// TwinCAT 3 PLC project TwinCAT_3_Program
// ProgramVersion: 3.1.4024.0
// libraries:
//   CmpBitmapPool, * (System)
//   Recipe Management, * (System)
//   Tc2_ControllerToolbox, * (Beckhoff Automation GmbH)
//   Tc2_Drive, * (Beckhoff Automation GmbH)
//   Tc2_EtherCAT, * (Beckhoff Automation GmbH)
//   Tc2_IoFunctions, * (Beckhoff Automation GmbH)
//   Tc2_Math, * (Beckhoff Automation GmbH)
//   Tc2_MC2, * (Beckhoff Automation GmbH)
//   Tc2_MC2_Drive, * (Beckhoff Automation GmbH)
//   Tc2_ModbusRTU, * (Beckhoff Automation GmbH)
//   Tc2_ModbusSrv, * (Beckhoff Automation GmbH)
//   Tc2_SerialCom, * (Beckhoff Automation GmbH)
//   Tc2_Standard, * (Beckhoff Automation GmbH)
//   Tc2_SUPS, * (Beckhoff Automation GmbH)
//   Tc2_System, * (Beckhoff Automation GmbH)
//   Tc2_Utilities, * (Beckhoff Automation GmbH)
//   Tc2_XmlDataSrv, * (Beckhoff Automation GmbH)
//   Tc3_Module, * (Beckhoff Automation GmbH)
//   VisuDialogs, * (System)
//   VisuSymbols,3.5.10.0,System
// project tree:
//   DUTs/DS TBD/ DSA1_ArmHorzPosInput.TcDUT, DSA1_ArmHorzPosOutput.TcDUT, DSA1_ArmPnpSequenceCall.TcDUT, DSA1_fbPnpSequenceMemoryCall.TcDUT, DSA1_fbPnpSequenceMemoryStore.TcDUT, DSA1_PnpSequenceMemory.TcDUT, DSA1_UpDownMovement.TcDUT, DSA21_UpDownPatternCall.TcDUT, DSA21_UpDownPatternMemory.TcDUT, DSA21_UpDownPatternStore.TcDUT, DSA31_ArmSpeedProfileCall.TcDUT, DSA31_ArmSpeedProfileMemory.TcDUT, DSA31_ArmSpeedProfileStore.TcDUT, DSA32_StationZoneHeight.TcDUT, DSA32_StationZoneHeightIntNotInUsed.TcDUT, DSA32_StationZonePosOut.TcDUT, DSChemicalWithoutDosingPump.TcDUT, DSGnr_CalledArmPnpParameter.TcDUT, DSPnpAgitationParameter.TcDUT, DSV2_A1_ArmHorzPosInput.TcDUT, DSV2_A1_ArmHorzPosOutput.TcDUT, DSV2_A1_ArmPnpSequenceCall.TcDUT, DSV2_A1_fbPnpSequenceMemoryCall.TcDUT, DSV2_A1_fbPnpSequenceMemoryStore.TcDUT, DSV2_A1_PnpSequenceMemory.TcDUT, DSV2_ApolloRemoteHoistInput.TcDUT, DSV2_ApolloRemoteHoistOutput.TcDUT, DSV2_ArmPosition.TcDUT, DSV2_BasketInfo.TcDUT, DSV2_ClangsonicGenerator.TcDUT, DSV2_fbGnrProductRecipeMemoryOut.TcDUT, DSV2_fbStationSequenceRecipeCall.TcDUT, DSV2_fbStationSequenceRecipeStore.TcDUT, DSV2_Gnr_CalledArmPnpParameter.TcDUT, DSV2_MinMaxEffTime.TcDUT, DSV2_ModbusControl.TcDUT, DSV2_SSERSourceMinMaxTime.TcDUT, DSV2_StationSequenceRecipeMemory.TcDUT, DSV2_StnMinMaxEffTIme.TcDUT, DSV2_TimeTrackerInput.TcDUT, DSV3_BarcodeRegistration.TcDUT, DSV3_JRS_Alarm.TcDUT, DSV3_JRS_HMI.TcDUT, DSV3_JRS_Input.TcDUT, DSV3_JRS_Output.TcDUT, DSV3_StnInterlock.TcDUT, DSV3_TempCtrlParameter.TcDUT, DSV3_TempCtrlRecipe.TcDUT, DSV3_XML_Recipe.TcDUT, DS_ArmPnPInOut.TcDUT, DS_BasketInfo.TcDUT, DS_BrensonEnclosure.TcDUT, DS_BrensonGenerator.TcDUT, DS_BrensonMulFreqSwitching.TcDUT, DS_ClangsonicGenerator.TcDUT, DS_fbGnrProductRecipeMemoryOut.TcDUT, DS_fbStationSequenceRecipeCall.TcDUT, DS_fbStationSequenceRecipeStore.TcDUT, DS_fbStationSubRecipeCall.TcDUT, DS_fbStationSubRecipeStore.TcDUT, DS_fbStnSeqProcessCtrl.TcDUT, DS_HMIStationDisplayInfo.TcDUT, DS_HomingSetting.TcDUT, DS_Inverter.TcDUT, DS_ProminentDosingHMI.TcDUT, DS_SA_Movement.TcDUT, DS_Servo.TcDUT, DS_StationSequenceRecipeMemory.TcDUT, DS_StnSeqProInput.TcDUT, DS_StnSeqProOutput.TcDUT, DS_SubRecipeMemory.TcDUT, DS_TimeTrackerInput.TcDUT, DS_WeberEnclosure.TcDUT, DS_WeberGenerator.TcDUT, DS_WeberMulFreqSwitching.TcDUT, DS_XMLRW.TcDUT, DS_XML_InputOutput.TcDUT, En_LogFileType.TcDUT, En_TimeInterval.TcDUT
//   DUTs/DS Twincat 3/Barcode/ DS_SerialCommunication.TcDUT
//   DUTs/DS Twincat 3/CSV/ DS_CsvErrorLog.TcDUT, DS_CsvLog.TcDUT, DS_CsvReport.TcDUT, E_CsvActionType.TcDUT
//   DUTs/DS Twincat 3/ DS_HMI_MappingVariable.TcDUT, DS_LocalSystemTime.TcDUT, DS_XML_Persistent_Analog.TcDUT, DS_XML_Persistent_Arm.TcDUT, DS_XML_Persistent_Barcode.TcDUT, DS_XML_Persistent_Deactivate.TcDUT, DS_XML_Persistent_Digital.TcDUT, DS_XML_Persistent_Memory.TcDUT, DS_XML_Persistent_Process.TcDUT, DS_XML_Persistent_SevenDay.TcDUT, DS_XML_Persistent_TimeOptimize.TcDUT, E_HmiLanguage.TcDUT, ST_DataLog.TcDUT
//   DUTs/DS Twincat 3/Enum/ Digital_Input.TcDUT, Digital_Output.TcDUT, Enum_Alarm_Others.TcDUT
//   DUTs/DS Twincat 3/Event/ DS_ActiveEventDisplay.TcDUT, DS_Event.TcDUT, DS_EventControl.TcDUT, DS_EventDescriptionCausedRemedy.TcDUT, DS_EventHistory.TcDUT, DS_EventHistoryLogToFile.TcDUT, DS_HistoryEventDisplay.TcDUT, E_EventType.TcDUT
//   DUTs/DS Twincat 3/UserCtrl/ DS_HmiUserReg.TcDUT, DS_HmiUserStatus.TcDUT, DS_VisuElement.TcDUT, eActorType.TcTLEO
//   DUTs/DS Twincat 3/XML/ E_XmlParType.TcDUT, E_XmlRwMode.TcDUT, E_XmlVariableType.TcDUT
//   FBs/B_JKS_CustomFB/fbArmCtrlFolder/ AM_MoveAbsolute.TcPOU, fbArmMoveInterLock.TcPOU, fbArmPnpCtrl.TcPOU, fbAxisPosCtrl.TcPOU, fbGenerateArmPickTransferBit.TcPOU, fbIndMotDecCtrl.TcPOU, fbInverterHorzHome.TcPOU, fbInverterJogCtrl.TcPOU, fbInverterPosCtrl.TcPOU, fbInverterVertHome.TcPOU, fbMotorHomingAxis.TcPOU, fbMultipleArmAgiCtrl.TcPOU, fbServoPosCmp.TcPOU, fbSlowPullAxisCtrl.TcPOU, fb_AxisMovement_Down.TcPOU, fb_AxisMovement_Up.TcPOU, FB_DRIVE_STATUS_ONE_AX.TcPOU
//   FBs/B_JKS_CustomFB/fbBarcodeCtrl/ fbBarcodeScanner.TcPOU, fbBarcodeSorting_10ML5575.TcPOU, fbBarcodeTracer.TcPOU, fbBarcodeTrancerNoCode.TcPOU, fbPreSuffixEliminator.TcPOU
//   FBs/B_JKS_CustomFB/fbConversionCtrl/ AM_InverterConversionHz.TcPOU, fbKeyenceVacSensorTuningkPa.TcPOU, fbRawRatioConversionAllenINV.TcPOU, fbRawRatioConversionReal.TcPOU, fbRawRatioConversionUs.TcPOU, fbRawRatioConversionUsPercent.TcPOU
//   FBs/B_JKS_CustomFB/fbDataLogCtrl/ FB_jx_DataLog.TcPOU, FB_TimeTriggering.TcPOU, FB_WriteLog.TcPOU, F_jx_TS_TO_DATE_STRING.TcPOU, F_jx_TS_TO_DATE_STRING_1.TcPOU, F_jx_TS_TO_TIME_STRING.TcPOU
//   FBs/B_JKS_CustomFB/fbGeneralfbFolder/ fbAssignBadBstCtrl.TcPOU, fbSlidingDoorCtrl.TcPOU, fbToleranceTimeCtrl.TcPOU, UserlevelFB.TcPOU
//   FBs/B_JKS_CustomFB/fbStnDegassingCtrl/ fbStnDegassCtrl.TcPOU
//   FBs/B_JKS_CustomFB/fbUltrasonicCtrl/ BrensonFreqSelector.TcPOU, fbUltrasonicFIFO.TcPOU, fbWeberUS_AI_Conversion.TcPOU, FB_WEBER.TcPOU, WeberFreqSelector.TcPOU
//   FBs/B_JKS_CustomFB/Other/ DoorOpenBasketTransfer.TcPOU, fbConveyorCtrl.TcPOU, fbIndirectAddStringArray.TcPOU, fbKeyConversionBarKpa.TcPOU, fbLdConveyor3Zones.TcPOU, fbLoadingConveyor3Zones.TcPOU, fbMultipleArmBasketMemory.TcPOU, fbPX3524ConversionBarKpa.TcPOU, fbStnRecipeWithSubAndCall.TcPOU, fbUld3ZoneConveyorCtrl.TcPOU, fbUldConveyor3Zones.TcPOU, fb_ArmBasketRotateCtrl.TcPOU, fb_StnCylinderInOutCtrl.TcPOU, HoldingBitSV.TcPOU, ReservoirTankDrain.TcPOU, ReservoirTankDrainNIL.TcPOU, TactTimeFB.TcPOU
//   FBs/B_JKS_NewFB/FBP-AlarmAndEvent/ fbAlarmModule.TcPOU
//   FBs/B_JKS_NewFB/FBP-ArmRelated/ fbA1_ArmHorzPosMemory.TcPOU, fbFBPArmHorzZoneConfirm.TcPOU, fbFBPVertArmPosConfirm.TcPOU, fbGnrProductRecipeMemory.TcPOU
//   FBs/B_JKS_NewFB/FBP-BasketTotalizer/ fbBasketTotalizer.TcPOU, fbStnBasketTotalizer.TcPOU
//   FBs/B_JKS_NewFB/FBP-EncoderIncrementalCtrl/ fbEncoderConversion.TcPOU
//   FBs/B_JKS_NewFB/FBP-HMIAddMapping/ fbHMIAddMappingArrayBool.TcPOU, fbHMIAddMappingArrayInt.TcPOU, fbHMIAddMappingArrayLreal.TcPOU, fbHMIAddMappingArrayReal.TcPOU, fbHMIAddMappingArrayString.TcPOU, fbHMIAddMappingBool.TcPOU, fbHMIAddMappingBoolForManual.TcPOU, fbHMIAddMappingDWordToBoolForManual.TcPOU, fbHMIAddMappingInt.TcPOU, fbHMIAddMappingInt_Word.TcPOU, fbHMIAddMappingLreal.TcPOU, fbHMIAddMappingReal.TcPOU, fbHMIAddMappingReal_Int.TcPOU, fbHMIAddMappingReal_Word.TcPOU, fbHMIAddMappingString.TcPOU
//   FBs/B_JKS_NewFB/FBP-HMI/ fbHMISimulateArmMovement.TcPOU, fbScrMapping.TcPOU
//   FBs/B_JKS_NewFB/FBP-Instrument/ fbBrensonMultiFreqCtrl.TcPOU, fbClangsonicUltrasonic.TcPOU, fbClangsonicUltrasonic_test.TcPOU, fbWeberMultiFreqCtrl.TcPOU
//   FBs/B_JKS_NewFB/FBP-MachineOperationTimeCounter/ fbMachineTimeCounter.TcPOU, fbVacuumPumpTimeCounter.TcPOU
//   FBs/B_JKS_NewFB/FBP-Memory_Sub/ fbA1_PnpSequenceMemory.TcPOU, fbA21_UpDownPattern.TcPOU, fbA31_ArmSpeedProfileMemory.TcPOU, fbA32_MachineZoneHeight.TcPOU, fbA32_StationZoneHeight.TcPOU, fbCallStnSeqSubPro.TcPOU, fbGnrStationMasterController.TcPOU, fbSingleArmBasketMemoryV2.TcPOU, fbStationSequenceRecipe.TcPOU, fbStationSubRecipe.TcPOU, fbStnSeqProcess.TcPOU
//   FBs/B_JKS_NewFB/FBP-ProcessOptimisation/ fbFBPTimeTrackerG2.TcPOU, fbFBPTimeTrackerG3.TcPOU, fbMasterTimeBlockG2.TcPOU, fbRecipeTimeBlockG2.TcPOU, fbTimeBlockSimulatorG2.TcPOU
//   FBs/B_JKS_NewFB/FBP-ProminentDosingPumpCtrl/ fbProminentDosingCtrl.TcPOU
//   FBs/B_JKS_NewFB/FBP-SevenDayAutoOnOff/ fbSevenDaySys.TcPOU
//   FBs/B_JKS_NewFB/FBP-StationRelated/ fbMainStationProcess.TcPOU
//   FBs/B_JKS_NewFB/FBP-TempController/ fbTempControl.TcPOU
//   FBs/B_JKS_NewFB/FBP-TowerLightCtrl/ fbTowerLightCtrl.TcPOU
//   FBs/B_JKS_NewFB_V2/fbArmCtrlFolder/ fbV2_1_ArmPnpCtrl.TcPOU
//   FBs/B_JKS_NewFB_V2/FBP-ArmCtrlFolder/ fbV2_ArmPnpCtrl.TcPOU, fbV2_GenerateArmPickTransferBit.TcPOU
//   FBs/B_JKS_NewFB_V2/FBP-ArmRelated/ fbV2_ArmPosSignalCtrl.TcPOU, fbV2_FBPArmHorzZoneConfirm.TcPOU, fbV2_GnrProductRecipeMemory.TcPOU, NIUfbV2_FBPVertArmPosConfirm.TcPOU
//   FBs/B_JKS_NewFB_V2/FBP-BasketInfoRelated/ fbV2_BasketInfoManager.TcPOU
//   FBs/B_JKS_NewFB_V2/FBP-Function_Sub/ fbAgitationCtrl.TcPOU, fbV2_BasketInfoFinder.TcPOU, fbV2_DSMovementHandler.TcPOU, fbV2_InvAnalogSpdCtrl.TcPOU, fbV2_InvAxisHome.TcPOU, fbV2_InvAxisJog.TcPOU, fbV2_InvPosCtrl.TcPOU
//   FBs/B_JKS_NewFB_V2/FBP-HMI/ fbV2_ScrMapping.TcPOU
//   FBs/B_JKS_NewFB_V2/FBP-Instrument/Dryer/ fbV2_DryerCoolingCtrl.TcPOU (not stored)
//   FBs/B_JKS_NewFB_V2/FBP-LdUldCVRelated/ fbV2_Cv2zonewith2m2sCtrl.TcPOU, fbV2_Cv3zonewith3m3sCtrl.TcPOU, fbV2_Cv4zonewith4m4sCtrl.TcPOU, fbV2_Cv5zonewith5m5sCtrl.TcPOU, fbV2_LdUldCvCtrl.TcPOU
//   FBs/B_JKS_NewFB_V2/FBP-Memory_Sub/ fbV2_A1_PnpSequenceMemory.TcPOU, fbV2_A32_MachineZoneHeight.TcPOU, fbV2_CallStnSeqSubPro.TcPOU, fbV2_GnrStationMasterController.TcPOU, fbV2_SingleArmBasketMemoryV2.TcPOU, fbV2_StationSequenceRecipe.TcPOU, fbV2_StnSeqProcess.TcPOU
//   FBs/B_JKS_NewFB_V2/FBP-MTBSubFB/ fbV2_HMIStnMinMaxEffTimeDisplay.TcPOU, fbV2_MinMaxExtShift.TcPOU, fbV2_SubAnalyzeRTBEffTime.TcPOU, fbV2_SubBusyRTBShifting.TcPOU, fbV2_SubFreeMTBShifting.TcPOU, fbV2_SubMTBFreeSlotGenerator.TcPOU, fbV2_SubMTBRTBCrashCheck.TcPOU, fbV2_SubMTBRunningTime.TcPOU, fbV2_SubRTBBusyLinkMTSUpdate.TcPOU, fbV2_SubRTBEndStepFinder.TcPOU, fbV2_SubRTBGenerateNoCallArmTime.TcPOU, fbV2_SubRTBStnTypeAltIDFinder.TcPOU, fbV2_SubTimeBlockCompare.TcPOU
//   FBs/B_JKS_NewFB_V2/FBP-ProcessOptimisation/ fbV2_FBPTimeTrackerG3.TcPOU, fbV2_MasterTimeBlockG2.TcPOU, fbV2_TimeBlockSimulatorG2.TcPOU
//   FBs/B_JKS_NewFB_V2/FBP-StationRelated/ fbV2_MainStationProcess.TcPOU
//   FBs/B_JKS_NewFB_V2/FBP-TempController/ fbV2_TempControl.TcPOU
//   FBs/B_JKS_NewFB_V3/CSV/ FB3_CsvHandler.TcPOU
//   FBs/B_JKS_NewFB_V3/Event/ FB3_EventModule.TcPOU
//   FBs/B_JKS_NewFB_V3/FBP-Memory_Sub/ fbV3_TemperatureParaRecipe.TcPOU
//   FBs/B_JKS_NewFB_V3/UserCtrl/ FB3_HmiTF1800_UserlevelManagement.TcPOU
//   FBs/B_JKS_NewFB_V3/XML/ FB3_XmlSvrRW_MultipleGVL.TcPOU, FB3_XmlSvrRW_Recipe.TcPOU
//   FBs/B_JKS_OldFB/Compare/ EQ_GT.TcPOU, EQ_LT.TcPOU, LT_GT.TcPOU, MANUAL_PAGE.TcPOU, SERVO_POS_CONFIRM.TcPOU
//   FBs/B_JKS_OldFB/Controller/ GUYSON_PRG_SEL.TcPOU, MOTION_ACC_DCC.TcPOU, TEMP_CTRL_ON_OFF.TcPOU, TEMP_CTRL_ON_OFF_EXT.TcPOU
//   FBs/B_JKS_OldFB/Converter/ DC_PID_FB.TcPOU, JOG_CONV.TcPOU, MM_TO_PLS.TcPOU
//   FBs/B_JKS_OldFB/Guyson/ GUYSON_AI_CTRL.TcPOU, GUYSON_AI_RawToWatt.TcPOU, GUYSON_AI_WattToRaw.TcPOU
//   FBs/B_JKS_OldFB/Memory/ INDIRECT_FN.TcPOU
//   FBs/B_JKS_OldFB/Timer/ CLOCK_PLS.TcPOU, DOWN_COUNT_TIMER.TcPOU, fbHoldingTimer.TcPOU, MOTION_COUNTER_RESET.TcPOU, TIMER_ALARM.TcPOU
//   FBs/B_JKS_OldFB/Word to Bit/ CMP_OC_DINT.TcPOU, CMP_OC_DW.TcPOU, CMP_OC_W1.TcPOU, CMP_OC_W10.TcPOU, CMP_OC_W2.TcPOU, CMP_OC_W3.TcPOU, CMP_OC_W4.TcPOU, CMP_OC_W5.TcPOU, CMP_OC_W6.TcPOU, CMP_OC_W7.TcPOU, CMP_OC_W8.TcPOU, CMP_OC_W9.TcPOU
//   FBs/b_JKS_RecycleFB/ fb_V3JRSModuleWithChiller.TcPOU
//   FBs/fbV3BarcodeCtrl/Main FB/ fb_V3BarcodeMasterCtrl.TcPOU
//   FBs/fbV3BarcodeCtrl/Sub FB/ fb_V1BarcodeRegistration_UTAC.TcPOU, fb_V2BarcodeRegistration.TcPOU, fb_V3BarcodeRegSectionDisplayController.TcPOU, fb_V3BarcodeScanner.TcPOU, fb_V3BarcodeTracer.TcPOU, fb_V3StringEliminator.TcPOU
//   FBs/FB_Others TBD/ fbArmSpecialFunctionStore.TcPOU, fbChemicalMixingWithoutPump.TcPOU, fbDetergent_BasketQuantityResetPB_PasswordControl.TcPOU, fbMapMobbusTCP.TcPOU, fbOilSeperatorTankCtrl.TcPOU, fbV3_ImportExportXML.TcPOU, fbV3_LoadingRecipeCheck.TcPOU, fbV3_TotalProcessTimeTracker.TcPOU, fbV3_XML_Handler.TcPOU, PID_FB.TcPOU
//   / GlobalTextList.TcGTLO, PlcTask.TcTTO, Visualization Manager.TcVMO (not stored)
//   GVLs/Alarm_Ctrl/ Global_Variables_Alarm.TcGVL
//   GVLs/Analog_Ctrl/ Global_Variables_Analog_NoPersistent.TcGVL, Global_Variables_Analog_Persistent.TcGVL, Global_Variables_DeclarationOnly.TcGVL
//   GVLs/Arm_Ctrl/ Global_Variables_Arm1BoolCtrl.TcGVL, Global_Variables_Arm2BoolCtrl.TcGVL, Global_Variables_Arm_NoPersistent.TcGVL, Global_Variables_Arm_Persistent.TcGVL
//   GVLs/Barcode_Ctrl/ Global_Variables_Barcode.TcGVL, Global_Variables_V3BarcodeScanner.TcGVL
//   GVLs/Constant_Ctrl/Constant_TC3/CONSTANT/ LIB_GVL_EVENT_CONSTANT.TcGVL (not stored), LIB_GVL_GENERAL_CONSTANT.TcGVL (not stored), LIB_GVL_IO_CONSTANT.TcGVL, LIB_GVL_MEMORY_CONSTANT.TcGVL (not stored)
//   GVLs/Constant_Ctrl/ Global_Variables_Constant.TcGVL
//   GVLs/Digital_Ctrl/ Global_Variables_DigitalBoolCtrl.TcGVL, Global_Variables_DigitalMapping.TcGVL, Global_Variables_Digital_Persistent.TcGVL
//   GVLs/General_Ctrl/ Global_Variables.TcGVL, Global_Variables_General_Fix.TcGVL, Global_Variables_General_Persistent.TcGVL
//   GVLs/GVL3/ GVL_Analog.TcGVL, GVL_Deactivate_Persistent.TcGVL, GVL_Event_Module.TcGVL, LIB_GVL_EVENT.TcGVL, LIB_GVL_GENERAL.TcGVL, LIB_GVL_IO.TcGVL, LIB_GVL_MEMORY.TcGVL
//   GVLs/HMI_Ctrl/ Global_Variables_CT12_HMIfunction.TcGVL, Global_Variables_HMI.TcGVL, Global_Variables_HMI_Function.TcGVL
//   GVLs/Internal Address/ GVL_Internal_Variable.TcGVL
//   GVLs/Memory_Ctrl/ Global_Variables_Memory.TcGVL
//   GVLs/ModbusTCP_Ctrl/ Global_Variables_Modbus.TcGVL
//   GVLs/Others TBD/ Globale_VarCheck.TcGVL, Global_HMI.TcGVL, Global_Variables_Lib_NonPresistent.TcGVL, Global_Variables_Lib_Persistent.TcGVL, Global_Variables_PID.TcGVL, Global_Variables_PID_1.TcGVL, GVL_HMI_CKK.TcGVL
//   GVLs/PDF_Report/ Global_Variables_PDF_Report.TcGVL
//   GVLs/Process_Ctrl/ Global_Variables_Process_NoPersistent.TcGVL, Global_Variables_Process_Persistent.TcGVL
//   GVLs/RecycleMachineJRSCtrl/ Global_Variables_JRS_HMI.TcGVL, Global_Variables_RecycleJRS.TcGVL
//   GVLs/Secs_Gem/ Global_Secs_Gem.TcGVL, Global_Variables_Secs_Gem_Persistent.TcGVL
//   GVLs/SevenDay_Ctrl/ Global_Variables_Process_Door.TcGVL, Global_Variables_SevenDay_NoPersistent.TcGVL, Global_Variables_SevenDay_Persistent.TcGVL
//   GVLs/Special_Ctrl/ Global_Variables_Special_NoPersistent.TcGVL, Global_Variables_Special_Persistent.TcGVL
//   GVLs/TimeOptimize_Ctrl/ Global_Variables_TimeOptimize.TcGVL
//   GVLs/UserCtrl/ GVL_UserCtrl.TcGVL
//   GVLs/XML_Ctrl/ XML.TcGVL
//   POUs/ MAIN.TcPOU
//   POUs/MainProgram/Aa_HmiVariableCtrl/ HMIValueKeyInCtrl.TcPOU
//   POUs/MainProgram/AgitationMechanismCtrl/ AgitationMechanismCtrl.TcPOU
//   POUs/MainProgram/AlertCtrl/ Alarm_IO.TcPOU, Alarm_Others.TcPOU, DeactivateCtrl.TcPOU, MisshookSensorCtrl.TcPOU
//   POUs/MainProgram/AnalogCtrl/ClangsonicUltrasonicCtrl/ ClangsonicUSCommCtrl.TcPOU (not stored), ClangsonicUSCtrl.TcPOU (not stored), ClangsonicUSModbusCtrl.TcPOU (not stored), ClangsonicUSModbusFeedbackCtrl.TcPOU (not stored), ModbusControl_ST.TcPOU (not stored)
//   POUs/MainProgram/AnalogCtrl/ConductivityCtrl/ ConductivityCtrl.TcPOU (not stored)
//   POUs/MainProgram/AnalogCtrl/FilterPressureCtrl/ FilterPressureCtrl.TcPOU (not stored)
//   POUs/MainProgram/AnalogCtrl/MegasonicCtrl/ MegasonicModbusProgram_ST.TcPOU (not stored)
//   POUs/MainProgram/AnalogCtrl/ Modbus_test.TcPOU
//   POUs/MainProgram/AnalogCtrl/TemperatureCtrl/ FBV4_PID.TcPOU (not stored), PID_ctrl.TcPOU (not stored), PID_ctrl_IR_Heater.TcPOU (not stored), PID_Ctrl_Test.TcPOU (not stored), PID_Difference_ctrl.TcPOU (not stored), PID_TempCtrl.TcPOU (not stored), TempChillerCtrl.TcPOU (not stored), TempCtrl.TcPOU (not stored)
//   POUs/MainProgram/AutoArmCtrl/ AxisHorzMovementOutputCtrl_Arm1.TcPOU, AxisServoCtrlMapping_Arm1.TcPOU, AxisServoCtrl_Arm1.TcPOU, AxisVertMovementOutputCtrl_Arm1.TcPOU, OmronServoEnable.TcPOU, PnpCtrl_Arm1.TcPOU, PnpMapping_Arm1.TcPOU, PnPstorageMemory_Arm.TcPOU, PosConfirmBitCtrl_Arm1.TcPOU
//   POUs/MainProgram/AutoArmCtrl/CoeRead/ HorzCoERead.TcPOU (not stored), SlowpullCoERead.TcPOU (not stored), VertCoERead.TcPOU (not stored)
//   POUs/MainProgram/AutoArmCtrl/Slowpull/ AxisHorzAdditionalInterlock_Arm1.TcPOU (not stored), AxisServoCtrl_SlowPull.TcPOU (not stored), oArmSlowPullHomingCtrl.TcPOU (not stored), oArmSlowPullOutputCtrl.TcPOU (not stored), PosConfirmBitCtrl_SlowPull.TcPOU (not stored)
//   POUs/MainProgram/AutoProcessCtrl/AutoModeProcessCtrl/ Cascading.TcPOU (not stored), StnOverflowValveCtrl.TcPOU (not stored)
//   POUs/MainProgram/AutoProcessCtrl/AutoModeProcessCtrl/Ld/ LdBasketMissingCtrl.TcPOU (not stored), LdPrcs.TcPOU (not stored), LdPrcs_General.TcPOU (not stored)
//   POUs/MainProgram/AutoProcessCtrl/AutoModeProcessCtrl/Process_Stn10/ Stn10.TcPOU (not stored)
//   POUs/MainProgram/AutoProcessCtrl/AutoModeProcessCtrl/Process_Stn1/ Stn1.TcPOU (not stored)
//   POUs/MainProgram/AutoProcessCtrl/AutoModeProcessCtrl/Process_Stn2/ Stn2.TcPOU (not stored)
//   POUs/MainProgram/AutoProcessCtrl/AutoModeProcessCtrl/Process_Stn3/ Stn3.TcPOU (not stored)
//   POUs/MainProgram/AutoProcessCtrl/AutoModeProcessCtrl/Process_Stn4/ Stn4.TcPOU (not stored)
//   POUs/MainProgram/AutoProcessCtrl/AutoModeProcessCtrl/Process_Stn5/ Stn5.TcPOU (not stored)
//   POUs/MainProgram/AutoProcessCtrl/AutoModeProcessCtrl/Process_Stn6/ Stn6.TcPOU (not stored)
//   POUs/MainProgram/AutoProcessCtrl/AutoModeProcessCtrl/Process_Stn7/ Stn7.TcPOU (not stored), Stn7ReturnPumpCtrl.TcPOU (not stored)
//   POUs/MainProgram/AutoProcessCtrl/AutoModeProcessCtrl/Process_Stn8/ Stn8.TcPOU (not stored)
//   POUs/MainProgram/AutoProcessCtrl/AutoModeProcessCtrl/Process_Stn9/ Stn9.TcPOU (not stored), Stn9SlowPullCalculation.TcPOU (not stored)
//   POUs/MainProgram/AutoProcessCtrl/ BarcodeScanner.TcPOU
//   POUs/MainProgram/AutoSevenDayOnOffCtrl/ SevenDayCtrl.TcPOU, SevenDayOnOffConf.TcPOU
//   POUs/MainProgram/A_StandardStructureProgram/ stClockPulseBlink.TcPOU, stGetCurrentTime.TcPOU, stUPSStatusMonitoring.TcPOU, stWritePersistentData.TcPOU
//   POUs/MainProgram/Barcode/ BarcodeCtrl_Utac.TcPOU, Barcode_Reg.TcPOU, SerialCom.TcPOU
//   POUs/MainProgram/BaseWork/ TowerLightCtrl.TcPOU
//   POUs/MainProgram/BasketMemory_RecipeCtrl/ BasketBadCtrl.TcPOU, BasketMemoryCtrl.TcPOU, BasketToleranceCtrl.TcPOU, BskMemoryCtrl.TcPOU, CvMotorREFE.TcPOU
//   POUs/MainProgram/CheckBound/ CheckBounds.TcPOU, CheckDivByte.TcPOU, CheckDivDWord.TcPOU, CheckDivLreal.TcPOU, CheckDivReal.TcPOU, CheckRangeSigned.TcPOU, CheckRangeUnsigned.TcPOU
//   POUs/MainProgram/Csv/ Batch_Number_counter.TcPOU, Csv_Report_Ctrl.TcPOU, Csv_Report_Mapping.TcPOU
//   POUs/MainProgram/DataManagement/ ArmPickTransferCtrl_General.TcPOU, BasketTotalizer.TcPOU, MacOperationTimeCtrl.TcPOU, RTClockCtrl.TcPOU, StnBasketTotalizer.TcPOU
//   POUs/MainProgram/DataManagement_Barcode/ GeneratorComparison.TcPOU, Log_BasketTimeInOut.TcPOU, Log_Configuration.TcPOU, Log_Management.TcPOU
//   POUs/MainProgram/DosingPumpCtrl/ ManualDosingSTreset.TcPOU, Stn1DosingPumpCtrl.TcPOU, Stn3DosingPumpCtrl.TcPOU, Stn5DosingPumpCtrl.TcPOU
//   POUs/MainProgram/HMI/ HMI_CKK.TcPOU, HMI_Ctrl.TcPOU, StartStop.TcPOU
//   POUs/MainProgram/ManualCtrl/ ManualButtonCtrl.TcPOU, ManualCtrl.TcPOU, ManualCtrl_Arm.TcPOU, ManualLifterJog.TcPOU
//   POUs/MainProgram/Mapping/ Internal_Mapping.TcPOU, IO_Mapping.TcPOU
//   POUs/MainProgram/OPC_UA/ OPC_UA_MAP.TcPOU (excluded from build)
//   POUs/MainProgram/Other/ ArmXYPosAdjust.TcPOU, BeckhoffHMIMapping.TcPOU, ClockPulse10ms.TcPOU, HMI_Function.TcPOU, HMI_Invinsible_Ctrl.TcPOU, HMI_Page_Control.TcPOU, HoldingBitCtrl.TcPOU, HoldingBit_DoorTransfer.TcPOU, ProHMIMapping.TcPOU, TactTime.TcPOU, zHMIMaxMinLimit.TcPOU
//   POUs/MainProgram/OutputCtrl/ MAIN_Arm_Mapping.TcPOU (not stored), MP_1_Y100.TcPOU (not stored), MP_2_Y101.TcPOU (not stored), MP_3_Y102.TcPOU (not stored), MP_4_Y103.TcPOU (not stored), SP1_1_Y110.TcPOU (not stored), SP1_2_Y111.TcPOU (not stored), SP2_1_Y120.TcPOU (not stored), SP3_1_Y130.TcPOU (not stored), SP3_2_Y131.TcPOU (not stored), SP3_3_Y132.TcPOU (not stored), STN_TopUpCtrl.TcPOU (not stored)
//   POUs/MainProgram/TimeOptimize/ Optimizer_Monitor.TcPOU, TimeOptimizeCtrl.TcPOU (not stored), TimeTrackerCtrl.TcPOU (not stored)
//   POUs/MainProgram/User/ UserCtrl.TcPOU
//   POUs/MainProgram/XML/Additional/ FBV4_SingleFileImportExport.TcPOU (not stored), Manual_ImportExport_Others.TcPOU (not stored)
//   POUs/MainProgram/XML/ Bootup_Shutdown_ctrl.TcPOU, pouXMLRecipeTest.TcPOU, XML_PersistentCtrl.TcPOU (not stored)
//   POUs/MainProgram/zAutoMode/ AutoMain.TcPOU (not stored), AutoMain_AddON.TcPOU, AutoOriginCtrl.TcPOU (not stored), AutoPreparationCtrl.TcPOU (not stored), AutoPreparationCtrl_ST.TcPOU (not stored), AutoStartCtrl.TcPOU (not stored)
//   VISUs/ALARM/ Alarm_Page.TcVIS
//   VISUs/AUTO/Auto all stn popup/ Auto_General.TcVIS (not stored), Auto_Loading.TcVIS (not stored), Auto_Station01.TcVIS (not stored), Auto_Station02.TcVIS (not stored), Auto_Station03.TcVIS (not stored), Auto_Station04.TcVIS (not stored), Auto_Station05.TcVIS (not stored), Auto_Station06.TcVIS (not stored), Auto_Unloading.TcVIS (not stored)
//   VISUs/AUTO/Auto main popup/ Popup_AllInfo.TcVIS (not stored), Popup_ArmInfo.TcVIS (not stored), Popup_OriginStatus.TcVIS (not stored), Popup_OtherInfo.TcVIS (not stored), Popup_PreparationStatus.TcVIS (not stored), Popup_ProcessStatus.TcVIS (not stored)
//   VISUs/AUTO/ AutoMain_Page.TcVIS, Auto_AllStation.TcVIS
//   VISUs/BARCODE/ Barcode_Page.TcVIS, Popup_Barcode.TcVIS, Popup_Ld_Warning.TcVIS
//   VISUs/DEACTIVATED/ Deactivated_Page.TcVIS
//   VISUs/ GlobalTextList_1.TcGTLO, ImagePool.TcIPO (not stored), Popup_Machine.TcVIS, Popup_Machine_Manual.TcVIS, Popup_MenuPage.TcVIS, RecipeNo.TcTLO, TextList_1_20.TcTLO, TextList_1_20_Speed.TcTLO, TextList_AccessLevel.TcTLO, TextList_Arm_Setting.TcTLO, TextList_ManualPage.TcTLO, TextList_Recipe.TcTLO, TextList_SettingPage.TcTLO, TextList_SettingPage_2.TcTLO, TextList_StationInfoPage.TcTLO, Vertical_Arm_Traveling_Zone.TcVIS, Visualization.TcVIS
//   VISUs/IO MONITORING/ IO_Monitoring.TcVIS
//   VISUs/IO MONITORING/Popup_IO/ Popup_IOinput.TcVIS (not stored), Popup_IOoutput.TcVIS (not stored)
//   VISUs/MANUAL/Manual mode pop up/ Manual_General.TcVIS (not stored), Manual_Loading.TcVIS (not stored), Manual_Station01.TcVIS (not stored), Manual_Station02.TcVIS (not stored), Manual_Station03.TcVIS (not stored), Manual_Station04.TcVIS (not stored), Manual_Station05.TcVIS (not stored), Manual_Station06.TcVIS (not stored), Manual_Unloading.TcVIS (not stored), Popup_ArmControl.TcVIS (not stored), Popup_SlowpullJog.TcVIS (not stored)
//   VISUs/MANUAL/ Manual_AllStation.TcVIS, Manual_Page.TcVIS
//   VISUs/POPUP/ Manual_Exit_Popup.TcVIS, Popup_Parameter.TcVIS, Popup_Parameter_Saved.TcVIS, Vacuum_Calibration.TcVIS
//   VISUs/RECIPE/Recipe Popup SSUR/ Recipe_AllStation_SSUR.TcVIS (not stored), Recipe_Station01.TcVIS (not stored), Recipe_Station02.TcVIS (not stored), Recipe_Station03.TcVIS (not stored), Recipe_Station04.TcVIS (not stored), Recipe_Station05.TcVIS (not stored), Recipe_Station06.TcVIS (not stored), Recipe_Station10.TcVIS (not stored), Recipe_Station11.TcVIS (not stored), Recipe_Station12.TcVIS (not stored)
//   VISUs/RECIPE/Recipe Popup/ Popup_RecipeConfiguration.TcVIS (not stored), Popup_RecipeSSER.TcVIS (not stored)
//   VISUs/RECIPE/ RecipeConfiguration_Page.TcVIS, RecipeSSER_Page.TcVIS, RecipeSSUR_Page.TcVIS, Recipe_Page.TcVIS
//   VISUs/SETTING/ SettingArm_Page.TcVIS, SettingProcess_Page.TcVIS, Setting_Page.TcVIS
//   VISUs/USER_LOGIN/ Login_Page.TcVIS
//   VISUs/USER_SETTING/ AddNewUser_Page.TcVIS, Edit_User.TcVIS, UserSetting_Page.TcVIS

CONFIGURATION TwinCAT_3_Program
    RESOURCE PLC ON TwinCAT3
        TASK PlcTask(INTERVAL := T#10ms, PRIORITY := 20);
        PROGRAM MAIN WITH PlcTask : MAIN;
    END_RESOURCE
END_CONFIGURATION

// ---- DUTs/DS TBD/DSA1_ArmHorzPosInput.TcDUT
TYPE DSA1_ArmHorzPosInput : (*Full Occupied Byte = 500*)
STRUCT

	sReservedBool : STRING(50); (* Byte "n+0~n+99" *)

	lrCurrentPos : LREAL; (* Byte "n+100~n+107" *)
	lrTargetPos : LREAL; (* Byte "n+108~n+115" *)
	lrPosConfirmToleranceSV  : LREAL; (* Byte "n+116~n+123" *)
	lr2ndSpeedSV : LREAL; (* Byte "n+124~n+131" *)
	lrLdHookPos : LREAL; (* Byte "n+132~n+139" *)
	lrLdUnhookPos : LREAL; (* Byte "n+140~n+147" *)
	lrUldHookPos : LREAL; (* Byte "n+148~n+155" *)
	lrUldUnhookPos : LREAL; (* Byte "n+156~n+163" *)

	ARlrStnHookPos : ARRAY [0..iHorzArmPosArrayQty] OF LREAL; (* Byte "n+164~n+331" *)
	ARlrStnUnhookPos : ARRAY [0..iHorzArmPosArrayQty] OF LREAL; (* Byte "n+332~n+499" *)


END_STRUCT
END_TYPE

// ---- DUTs/DS TBD/DSA1_ArmHorzPosOutput.TcDUT
TYPE DSA1_ArmHorzPosOutput : (*Full Occupied Byte = 100*)
STRUCT

	bLdHookPosConfirm : BOOL; (* Byte "n" *)
	bLdUnhookPosConfirm : BOOL; (* Byte "n+1" *)
	bUldHookPosConfirm : BOOL; (* Byte "n+2" *)
	bUldUnhookPosConfirm : BOOL; (* Byte "n+3" *)
	ARbStnHookPosConfirm : ARRAY [0..iHorzArmPosArrayQty] OF BOOL; (* Byte "n+4 ~ Byte "n+24" *)
	ARbStnUnhookPosConfirm : ARRAY [0..iHorzArmPosArrayQty] OF BOOL; (* Byte "n+25 ~ Byte "n+45" *)

	bLdHook2ndSpeedEn : BOOL; (* Byte "n+46" *)
	bLdUnhook2ndSpeedEn : BOOL; (* Byte "n+47" *)
	bUldHook2ndSpeedEn : BOOL; (* Byte "n+48" *)
	bUldUnhook2ndSpeedEn : BOOL; (* Byte "n+49" *)
	ARbStnHook2ndSpeedEn : ARRAY [0..iHorzArmPosArrayQty] OF BOOL; (* Byte "n+50 ~ Byte "n+70" *)
	ARbStnUnhook2ndSpeedEn : ARRAY [0..iHorzArmPosArrayQty] OF BOOL; (* Byte "n+71 ~ Byte "n+91" *)
	sReservedBool : STRING(50); (* Byte "n+92~n+99" *)

END_STRUCT
END_TYPE

// ---- DUTs/DS TBD/DSA1_ArmPnpSequenceCall.TcDUT
TYPE DSA1_ArmPnpSequenceCall : (*Full Occupied Byte = 1700*)
STRUCT

	bEnableCallArmNo 					: BOOL; (* Byte "n" *)
	bCallSt								: BOOL; (* Byte "n+1" *)

	bCallCompleted 						: BOOL; (* Byte "n+2" *)
	bInvalidProductRecipeNoErrHold		: BOOL; (* Byte "n+3" *)
	bInvalidProductRecipeNoErrPulse	: BOOL; (* Byte "n+4" *)
	bInvalidProductRecipeStepErrHold 	: BOOL; (* Byte "n+5" *)
	bInvalidProductRecipeStepErrPulse	: BOOL; (* Byte "n+6" *)
	bCallUpDownPatternMemoryErr 		: BOOL; (* Byte "n+7" *)
	bCallArmSpeedProfileMemoryErr 	: BOOL; (* Byte "n+8" *)
	bCallPickStationNoErr 				: BOOL; (* Byte "n+9" *)
	bCallTransferStationNoErr 			: BOOL; (* Byte "n+10" *)

	sReservedBool 						: STRING(50); (* Byte "n+11~n+99" *)

	iCallArmNo 							: INT; (* Byte "n+100~n+101" *)
	iProductRecipeNoCall 				: INT; (* Byte "n+102~n+103" *)
	iProductRecipeStepCall				: INT; (* Byte "n+104~n+105" *)
	iCalledProductRecipeNo 				: INT; (* Byte "n+106~n+107" *) (*New*)
	iCalledProductRecipeStep			: INT; (* Byte "n+108~n+109" *) (*New*)

	sReservedInt 							: STRING(50); (* Byte "n+110~n+199" *)

	sProductRecipeDescription 			: STRING(50);


	DSGnrCalledArmPnpParameter 		: DSGnr_CalledArmPnpParameter;



END_STRUCT
END_TYPE

// ---- DUTs/DS TBD/DSA1_fbPnpSequenceMemoryCall.TcDUT
TYPE DSA1_fbPnpSequenceMemoryCall : (*Full Occupied Byte = 1100*)
STRUCT
	bCallPB: BOOL; (* Byte "n" *)
	bCallCompleted : BOOL; (* Byte "n+1" *)
	bInvalidCallProductRecipeNoHold : BOOL; (* Byte "n+2" *)
	bInvalidCallProductRecipeNoPulse : BOOL; (* Byte "n+3" *)
	sReservedBool : STRING(50); (* Byte "n+4~n+99" *)


	Call_iProductRecipeNo : INT; (* Byte "n+100, n+101" *)
	sReservedInt : STRING(50); (* Byte "n+102~n+199" *)


(*	Call_sSequenceRecipeDescription : STRING(50); (* Byte "n+200~n+299" *)*)
	sReserveString : STRING(50); (* Byte "n+200~n+299" *)

	Call_DsPnpSequenceMemory : DSA1_PnpSequenceMemory; (* Byte "n+300 onward" *)

END_STRUCT
END_TYPE

// ---- DUTs/DS TBD/DSA1_fbPnpSequenceMemoryStore.TcDUT
TYPE DSA1_fbPnpSequenceMemoryStore : (*Full Occupied Byte = 1100*)
STRUCT

	bCopyPB : BOOL; (* Byte "n" *)
	sReservedBool : STRING(98); (* Byte "n+1~n+99" *)


	iProductRecipeNo: INT; (* Byte "n+100, n+101" *)	(* 10 sets of Station Sequence Recipe *)
	iCopyToProductRecipeNo : INT; (* Byte "n+102, n+103" *)
	sReservedInt : STRING(95); (* Byte "n+104~n+199" *)


(*	sStationSequenceRecipeDescription : STRING(50); (* Byte "n+200~n+299" *)  (* Description of Station Sequence Recipe - Naming*)*)
	sReserveString : STRING(50); (* Byte "n+200~n+299" *)

	DsA1inPnpSequenceMemory : DSA1_PnpSequenceMemory; (* Byte "n+300 onward" *)


END_STRUCT
END_TYPE

// ---- DUTs/DS TBD/DSA1_PnpSequenceMemory.TcDUT
TYPE DSA1_PnpSequenceMemory : (*Full Occupied Byte = 800*)
STRUCT

	bZone1RepeatUpDnEnable : BOOL; (* Byte "n+0 *)
	bZone2RepeatUpDnEnable : BOOL; (* Byte "n+1 *)
	bZone3RepeatUpDnEnable : BOOL; (* Byte "n+2 *)
	bZone4RepeatUpDnEnable : BOOL; (* Byte "n+3 *)


	sReservedBool : STRING(95); (* Byte "n+4 ~ n+99" *)

	ARiCallArmNo : ARRAY [0..iProductRecipeStepArrayQty] OF INT; (* Byte "n+100~n+161" *)

	ARiPickStationNo : ARRAY [0..iProductRecipeStepArrayQty] OF INT; (* Byte "n+162~n+223" *)
	ARiTransferStationNo : ARRAY [0..iProductRecipeStepArrayQty] OF INT; (* Byte "n+224~n+285" *)

	ARiDownPickPatternNo : ARRAY [0..iProductRecipeStepArrayQty] OF INT; (* Byte "n+286~n+347" *)
	ARiUpPickPatternNo : ARRAY [0..iProductRecipeStepArrayQty] OF INT; (* Byte "n+348~n+409" *)
	ARiDownTransferPatternNo : ARRAY [0..iProductRecipeStepArrayQty] OF INT; (* Byte "n+410~n+471" *)
	ARiUpTransferPatternNo : ARRAY [0..iProductRecipeStepArrayQty] OF INT; (* Byte "n+472~n+533" *)

	ARiRepeatUpDownCycle : ARRAY [0..iProductRecipeStepArrayQty] OF INT; (* Byte "n+534~n+595" *)

	ARiStnSeqRepNo : ARRAY [0..iProductRecipeStepArrayQty] OF INT; (* Byte "n+596~n+657" *)

	sReservedInt : STRING(41); (* Byte "n+658~n+699" *)

	sDescription : STRING(50); (* Byte "n+700 ~ n+799" *)


END_STRUCT
END_TYPE

// ---- DUTs/DS TBD/DSA1_UpDownMovement.TcDUT
TYPE DSA1_UpDownMovement : (*Full Occupied Byte = 300*)
STRUCT
(*	sReservedBool : STRING(50); (* Byte "n+0 ~ n+99" *)*)
	lrZone1StartPos : LREAL; (* Byte "n+0~n+7" *)
	lrZone1EndPos : LREAL; (* Byte "n+8~n+15" *)
	lrZone2StartPos : LREAL; (* Byte "n+16~n+23" *)
	lrZone2EndPos : LREAL; (* Byte "n+24~n+31" *)
	lrZone3StartPos : LREAL; (* Byte "n+32~n+39" *)
	lrZone3EndPos : LREAL; (* Byte "n+40~n+47" *)
	lrZone4StartPos : LREAL; (* Byte "n+48~n+55" *)
	lrZone4EndPos : LREAL; (* Byte "n+56~n+63" *)


	lrZone1SpeedVelo : LREAL; (* Byte "64+0~n+71" *)
	lrZone2SpeedVelo : LREAL; (* Byte "72+0~n+79" *)
	lrZone3SpeedVelo : LREAL; (* Byte "80+0~n+87" *)
	lrZone4SpeedVelo : LREAL; (* Byte "88+0~n+95" *)

	lrZone1Acc : LREAL; (* Byte "n+96~n+103" *)
	lrZone1Dcc : LREAL; (* Byte "n+104~n+111" *)
	lrZone2Acc : LREAL; (* Byte "n+112~n+119" *)
	lrZone2Dcc : LREAL; (* Byte "n+120~n+127" *)
	lrZone3Acc : LREAL; (* Byte "n+128~n+135" *)
	lrZone3Dcc : LREAL; (* Byte "n+136~n+143" *)
	lrZone4Acc : LREAL; (* Byte "n+144~n+151" *)
	lrZone4Dcc : LREAL; (* Byte "n+152~n+159" *)

	lrMidPos		: LREAL; (* Byte "n+160~n+167" *) (*Added*)

	sReservedLreal : STRING(31); (* Byte "n+168~n+199" *)

	sUpDownPatternDescription : STRING(50); (* Byte "n+200 ~ n+299*)

END_STRUCT
END_TYPE

// ---- DUTs/DS TBD/DSA21_UpDownPatternCall.TcDUT
TYPE DSA21_UpDownPatternCall : (*Full Occupied Byte = 500*)
STRUCT
	bCallPB: BOOL; (* Byte "n" *)
	bCallCompleted : BOOL; (* Byte "n+1" *)
	bInvalidCallUpDownPatternNoHold : BOOL; (* Byte "n+2" *)
	bInvalidCallUpDownPatternNoPulse : BOOL; (* Byte "n+3" *)
	sReservedBool : STRING(95); (* Byte "n+4~n+99" *)


	Call_iUpDownPatternNo : INT; (* Byte "n+100, n+101" *)
	sReservedInt : STRING(97); (* Byte "n+102~n+199" *)


(*	Call_sSequenceRecipeDescription : STRING(50); (* Byte "n+200~n+299" *)*)


	Call_DsUpDownPattern : DSA21_UpDownPatternMemory; (* Byte "n+200 onward" *)

END_STRUCT
END_TYPE

// ---- DUTs/DS TBD/DSA21_UpDownPatternMemory.TcDUT
TYPE DSA21_UpDownPatternMemory : (*Full Occupied Byte = 300*)
STRUCT

	sReservedBool : STRING(50); (* Byte "n+0 ~ n+99" *)

	iZone1SpdProfileNo : INT; (* Byte "n+100, n+101" *)
	iZone2SpdProfileNo : INT; (* Byte "n+102, n+103" *)
	iZone3SpdProfileNo : INT; (* Byte "n+104, n+105" *)
	iZone4SpdProfileNo : INT; (* Byte "n+106, n+107" *)

	sReservedInt : STRING(91); (* Byte "n+108~n+199" *)



	sDescription : STRING(50); (* Byte "n+200 ~ n+299" *)


END_STRUCT
END_TYPE

// ---- DUTs/DS TBD/DSA21_UpDownPatternStore.TcDUT
TYPE DSA21_UpDownPatternStore : (*Full Occupied Byte = 500*)
STRUCT

	bCopyPB : BOOL; (* Byte "n" *)
	sReservedBool : STRING(98); (* Byte "n+1~n+99" *)


	iUpDownPatternNo: INT; (* Byte "n+100, n+101" *)	(* 10 sets of Station Sequence Recipe *)
	iCopyToUpDownPatternNo : INT; (* Byte "n+102, n+103" *)
	sReservedInt : STRING(95); (* Byte "n+104~n+199" *)


(*	sStationSequenceRecipeDescription : STRING(50); (* Byte "n+200~n+299" *)  (* Description of Station Sequence Recipe - Naming*)*)


	DsInUpDownPatternMemory : DSA21_UpDownPatternMemory; (* Byte "n+200 onward" *)


END_STRUCT
END_TYPE

// ---- DUTs/DS TBD/DSA31_ArmSpeedProfileCall.TcDUT
TYPE DSA31_ArmSpeedProfileCall : (*Full Occupied Byte = 500*)
STRUCT
	bCallPB: BOOL; (* Byte "n" *)
	bCallCompleted : BOOL; (* Byte "n+1" *)
	bInvalidCallArmSpdProfileNoHold : BOOL; (* Byte "n+2" *)
	bInvalidCallArmSpdProfileNoPulse : BOOL; (* Byte "n+3" *)
	sReservedBool : STRING(95); (* Byte "n+4~n+99" *)


	Call_iArmSpdProfile : INT; (* Byte "n+100, n+101" *)
	sReservedInt : STRING(97); (* Byte "n+102~n+199" *)


(*	Call_sSequenceRecipeDescription : STRING(50); (* Byte "n+200~n+299" *)*)


	Call_DSArmSpdProfile : DSA31_ArmSpeedProfileMemory; (* Byte "n+200 onward" *)

END_STRUCT
END_TYPE

// ---- DUTs/DS TBD/DSA31_ArmSpeedProfileMemory.TcDUT
TYPE DSA31_ArmSpeedProfileMemory : (*Full Occupied Byte = 300*)
STRUCT

	sReservedBool : STRING(50); (* Byte "n+0 ~ n+99" *)

(*	sReservedInt : STRING(49); (* Byte "n+100~n+149" *)*)

	lrSpeedVelo : LREAL; (* Byte "n+100~n+107" *)
	lrAcc : LREAL; (* Byte "n+108~n+115" *)
	lrDcc : LREAL; (* Byte "n+116~n+123" *)

	sReservedLreal : STRING(75); (* Byte "n+124~n+199" *)

	sDescription : STRING(50); (* Byte "n+200 ~ n+299" *)


END_STRUCT
END_TYPE

// ---- DUTs/DS TBD/DSA31_ArmSpeedProfileStore.TcDUT
TYPE DSA31_ArmSpeedProfileStore : (*Full Occupied Byte = 500*)
STRUCT

	bCopyPB : BOOL; (* Byte "n" *)
	sReservedBool : STRING(98); (* Byte "n+1~n+99" *)


	iArmSpdProfileNo: INT; (* Byte "n+100, n+101" *)	(* 10 sets of Station Sequence Recipe *)
	iCopyToSpdProfileNo : INT; (* Byte "n+102, n+103" *)
	sReservedInt : STRING(95); (* Byte "n+104~n+199" *)


(*	sStationSequenceRecipeDescription : STRING(50); (* Byte "n+200~n+299" *)  (* Description of Station Sequence Recipe - Naming*)*)


	DsArmSpeedProfile : DSA31_ArmSpeedProfileMemory; (* Byte "n+200 onward" *)


END_STRUCT
END_TYPE

// ---- DUTs/DS TBD/DSA32_StationZoneHeight.TcDUT
TYPE DSA32_StationZoneHeight : (*Full Occupied Byte = 200*)
STRUCT

	sReservedBool : STRING(50); (* Byte "n+0 ~ n+99" *)

(*	sReservedInt : STRING(49); (* Byte "n+100~n+149" *)*)

	lrTopPos : LREAL; (* Byte "n+100~n+107" *)
	lrZone1Range : LREAL; (* Byte "n+108~n+115" *)
	lrZone2Range : LREAL; (* Byte "n+116~n+123" *)
	lrZone3Range : LREAL; (* Byte "n+124~n+131" *)
	lrZone4Range : LREAL; (* Byte "n+132~n+139" *)
	lrBottomPos : LREAL; (* Byte "n+140~n+147" *)

	lrMidPos : LREAL; (*Byte "n+148~n+155*)

	sReservedLreal : STRING(43); (* Byte "n+156~n+199" *)

END_STRUCT
END_TYPE

// ---- DUTs/DS TBD/DSA32_StationZoneHeightIntNotInUsed.TcDUT
TYPE DSA32_StationZoneHeightIntNotInUsed : (*Full Occupied Byte = 200*)
STRUCT

	sReservedBool : STRING(50); (* Byte "n+0 ~ n+99" *)

(*	sReservedInt : STRING(49); (* Byte "n+100~n+149" *)*)

	lrTopPos : INT; (* Byte "n+100~n+101" *)
	lrZone1Range : INT; (* Byte "n+102~n+103" *)
	lrZone2Range : INT; (* Byte "n+104~n+105" *)
	lrZone3Range : INT; (* Byte "n+106~n+107" *)
	lrZone4Range : INT; (* Byte "n+108~n+109" *)
	lrBottomPos : INT; (* Byte "n+110~n+111" *)

	lrMidPos : INT; (*Byte "n+112~n+113*)

	sReservedLreal : STRING(85); (* Byte "n+114~n+199" *)

END_STRUCT
END_TYPE

// ---- DUTs/DS TBD/DSA32_StationZonePosOut.TcDUT
TYPE DSA32_StationZonePosOut : (*Full Occupied Byte = 200*)
STRUCT

	sReservedBool : STRING(50); (* Byte "n+0 ~ n+99" *)

(*	sReservedInt : STRING(49); (* Byte "n+110~n+149" *)*)

	lrZone1StartPos : LREAL; (* Byte "n+100~n+107" *)
	lrZone1EndPos : LREAL; (* Byte "n+108~n+115" *)
	lrZone2StartPos : LREAL; (* Byte "n+116~n+123" *)
	lrZone2EndPos : LREAL; (* Byte "n+124~n+131" *)
	lrZone3StartPos : LREAL; (* Byte "n+132~n+139" *)
	lrZone3EndPos : LREAL; (* Byte "n+140~n+147" *)
	lrZone4StartPos : LREAL; (* Byte "n+148~n+155" *)
	lrZone4EndPos : LREAL; (* Byte "n+156~n+163" *)

	lrMidPos : LREAL; (*Byte "n+164~n+171*)

	sReservedLreal : STRING(27); (* Byte "n+172~n+199" *)

END_STRUCT
END_TYPE

// ---- DUTs/DS TBD/DSChemicalWithoutDosingPump.TcDUT
TYPE DSChemicalWithoutDosingPump :
STRUCT

(*Input*)
	IN_b1StFillEnable						: BOOL;
	IN_bBasketResetQty					: BOOL;
	IN_i1stLimitBasketQty					: INT;
	IN_i2ndLimitBasketQty					: INT;
	IN_diMixingTime						: DINT;
	IN_bChemicalTopUpNotice				: BOOL;
	IN_bBasketCounterUp					: BOOL;

(*Output*)

	OUT_iCurrentBasketQty				: INT;
	OUT_b1stLimitBasketAlarm				: BOOL;
	OUT_b2ndLimitBasketAlarm			: BOOL;


	OUT_b1stFillChemicalTopUpBit			: BOOL;
	OUT_bProcessFillChemicalTopupBit		: BOOL;
	OUT_b1stFillCompleted				: BOOL;

END_STRUCT
END_TYPE

// ---- DUTs/DS TBD/DSGnr_CalledArmPnpParameter.TcDUT
TYPE DSGnr_CalledArmPnpParameter : (*Full Occupied Byte = 1400*)
STRUCT

	iCallArmNo : INT; (* Byte "n~, n+1" *)
	iStnSeqRecipeNo : INT; (* Byte "n+2, n+3" *)
	iPickStationNo : INT; (* Byte "n+4, n+5" *)
	iTransferStationNo : INT; (* Byte "n+6, n+7" *)

	iDrippingTimeSV : INT; (* Byte "n+8, n+9" *)

	sReservedInt : STRING(189); (* Byte "n+10~n+199" *)

	DSA1DownPickMovement : DSA1_UpDownMovement;
	DSA1UpPickMovement : DSA1_UpDownMovement;
	DSA1DownTransferMovement : DSA1_UpDownMovement;
	DSA1UpTransferMovement : DSA1_UpDownMovement;

END_STRUCT
END_TYPE

// ---- DUTs/DS TBD/DSPnpAgitationParameter.TcDUT
TYPE DSPnpAgitationParameter :
STRUCT

	bAgitationInProgress					: BOOL;
	bAgitationComplete					: BOOL;

	lrAgitationTopPosition					: LREAL;
	lrAgitationBtmPosition					: LREAL;

	bTopPositionCFM						: BOOL;
	bBtmPositionCFM						: BOOL;

	lrAgitationSpeed						: LREAL;
	lrAgitationSpeedAcc					: LREAL;
	lrAgitationSpeedDcc					: LREAL;

	iRepeatUpDownCycle					: INT;
	bPickRepeatStnEnable				: BOOL;
	bTransferRepeatStnEnable				: BOOL;

(*Output*)
(*
	iRepeatUpDownCycle					: INT;

	bPickRepeatStnEnable				: BOOL;
	bTransferRepeatStnEnable				: BOOL;
*)
	bSearchFinish						: BOOL;

END_STRUCT
END_TYPE

// ---- DUTs/DS TBD/DSV2_A1_ArmHorzPosInput.TcDUT
TYPE DSV2_A1_ArmHorzPosInput : (*Full Occupied Byte = 500*)
STRUCT

	sReservedBool 			: STRING(50); (* Byte "n+0~n+99" *)

	lrCurrentPos 				: LREAL; (* Byte "n+100~n+107" *)
	lrTargetPos 				: LREAL; (* Byte "n+108~n+115" *)
	lrPosConfirmToleranceSV  	: LREAL; (* Byte "n+116~n+123" *)
	lr2ndSpeedSV 			: LREAL; (* Byte "n+124~n+131" *)
	ARlrLdHookPos 			: ARRAY [0..iLdStnQty] OF LREAL; (* Byte "n+132~n+139" *)
	ARlrLdUnhookPos 		: ARRAY [0..iLdStnQty] OF LREAL; (* Byte "n+140~n+147" *)
	ARlrUldHookPos 			: ARRAY [0..iUldStnQty] OF LREAL; (* Byte "n+148~n+155" *)
	ARlrUldUnhookPos 		: ARRAY [0..iUldStnQty] OF LREAL; (* Byte "n+156~n+163" *)

	ARlrStnHookPos 			: ARRAY [0..iStnQty] OF LREAL; (* Byte "n+164~n+331" *)
	ARlrStnUnhookPos 		: ARRAY [0..iStnQty] OF LREAL; (* Byte "n+332~n+499" *)


END_STRUCT
END_TYPE

// ---- DUTs/DS TBD/DSV2_A1_ArmHorzPosOutput.TcDUT
TYPE DSV2_A1_ArmHorzPosOutput : (*Full Occupied Byte = 100*)
STRUCT

	ARbLdHookPosConfirm 			: ARRAY [0..iLdStnQty] OF BOOL; (* Byte "n" *)
	ARbLdUnhookPosConfirm		 	: ARRAY [0..iLdStnQty] OF BOOL; (* Byte "n+1" *)
	ARbUldHookPosConfirm 			: ARRAY [0..iUldStnQty] OF BOOL; (* Byte "n+2" *)
	ARbUldUnhookPosConfirm 			: ARRAY [0..iUldStnQty] OF BOOL; (* Byte "n+3" *)
	ARbStnHookPosConfirm 			: ARRAY [0..iStnQty] OF BOOL; (* Byte "n+4 ~ Byte "n+24" *)
	ARbStnUnhookPosConfirm 			: ARRAY [0..iStnQty] OF BOOL; (* Byte "n+25 ~ Byte "n+45" *)

	ARbLdHook2ndSpeedEn 			: ARRAY [0..iLdStnQty] OF BOOL; (* Byte "n+46" *)
	ARbLdUnhook2ndSpeedEn 		: ARRAY [0..iLdStnQty] OF BOOL; (* Byte "n+47" *)
	ARbUldHook2ndSpeedEn 			: ARRAY [0..iUldStnQty] OF BOOL; (* Byte "n+48" *)
	ARbUldUnhook2ndSpeedEn 		: ARRAY [0..iUldStnQty] OF BOOL; (* Byte "n+49" *)
	ARbStnHook2ndSpeedEn 			: ARRAY [0..iStnQty] OF BOOL; (* Byte "n+50 ~ Byte "n+70" *)
	ARbStnUnhook2ndSpeedEn 		: ARRAY [0..iStnQty] OF BOOL; (* Byte "n+71 ~ Byte "n+91" *)
	sReservedBool 					: STRING(7); (* Byte "n+92~n+99" *)

END_STRUCT
END_TYPE

// ---- DUTs/DS TBD/DSV2_A1_ArmPnpSequenceCall.TcDUT
TYPE DSV2_A1_ArmPnpSequenceCall : (*Full Occupied Byte = 1700*)
STRUCT

	bEnableCallArmNo 					: BOOL; (* Byte "n" *)
	bCallSt								: BOOL; (* Byte "n+1" *)

	bCallCompleted 						: BOOL; (* Byte "n+2" *)
	bInvalidProductRecipeNoErrHold		: BOOL; (* Byte "n+3" *)
	bInvalidProductRecipeNoErrPulse	: BOOL; (* Byte "n+4" *)
	bInvalidProductRecipeStepErrHold 	: BOOL; (* Byte "n+5" *)
	bInvalidProductRecipeStepErrPulse	: BOOL; (* Byte "n+6" *)
	bCallUpDownPatternMemoryErr 		: BOOL; (* Byte "n+7" *)
	bCallArmSpeedProfileMemoryErr 	: BOOL; (* Byte "n+8" *)
	bCallPickStationNoErr 				: BOOL; (* Byte "n+9" *)
	bCallTransferStationNoErr 			: BOOL; (* Byte "n+10" *)

	sReservedBool 						: STRING(88); (* Byte "n+11~n+99" *)

	iCallArmNo 							: INT; (* Byte "n+100~n+101" *)
	iProductRecipeNoCall 				: INT; (* Byte "n+102~n+103" *)
	iProductRecipeStepCall				: INT; (* Byte "n+104~n+105" *)
	iCalledProductRecipeNo 				: INT; (* Byte "n+106~n+107" *) (*New*)
	iCalledProductRecipeStep			: INT; (* Byte "n+108~n+109" *) (*New*)

	sReservedInt 							: STRING(89); (* Byte "n+110~n+199" *)

	sProductRecipeDescription 			: STRING(50);


	DSGnrCalledArmPnpParameter 		: DSV2_Gnr_CalledArmPnpParameter;



END_STRUCT
END_TYPE

// ---- DUTs/DS TBD/DSV2_A1_fbPnpSequenceMemoryCall.TcDUT
TYPE DSV2_A1_fbPnpSequenceMemoryCall : (*Full Occupied Byte = 1100*)
STRUCT
	bCallPB: BOOL; (* Byte "n" *)
	bCallCompleted : BOOL; (* Byte "n+1" *)
	bInvalidCallProductRecipeNoHold : BOOL; (* Byte "n+2" *)
	bInvalidCallProductRecipeNoPulse : BOOL; (* Byte "n+3" *)
	sReservedBool : STRING(95); (* Byte "n+4~n+99" *)


	Call_iProductRecipeNo : INT; (* Byte "n+100, n+101" *)
	sReservedInt : STRING(97); (* Byte "n+102~n+199" *)


(*	Call_sSequenceRecipeDescription : STRING(50); (* Byte "n+200~n+299" *)*)
	sReserveString : STRING(50); (* Byte "n+200~n+299" *)

	Call_DsPnpSequenceMemory : DSV2_A1_PnpSequenceMemory; (* Byte "n+300 onward" *)

END_STRUCT
END_TYPE

// ---- DUTs/DS TBD/DSV2_A1_fbPnpSequenceMemoryStore.TcDUT
TYPE DSV2_A1_fbPnpSequenceMemoryStore : (*Full Occupied Byte = 1100*)
STRUCT

	bCopyPB : BOOL; (* Byte "n" *)
	sReservedBool : STRING(98); (* Byte "n+1~n+99" *)


	iProductRecipeNo: INT; (* Byte "n+100, n+101" *)	(* 10 sets of Station Sequence Recipe *)
	iCopyToProductRecipeNo : INT; (* Byte "n+102, n+103" *)
	sReservedInt : STRING(95); (* Byte "n+104~n+199" *)


(*	sStationSequenceRecipeDescription : STRING(50); (* Byte "n+200~n+299" *)  (* Description of Station Sequence Recipe - Naming*)*)
	sReserveString : STRING(50); (* Byte "n+200~n+299" *)

	DsA1inPnpSequenceMemory : DSV2_A1_PnpSequenceMemory; (* Byte "n+300 onward" *)


END_STRUCT
END_TYPE

// ---- DUTs/DS TBD/DSV2_A1_PnpSequenceMemory.TcDUT
TYPE DSV2_A1_PnpSequenceMemory : (*Full Occupied Byte = 800*)
STRUCT

	bZone1RepeatUpDnEnable : BOOL; (* Byte "n+0 *)
	bZone2RepeatUpDnEnable : BOOL; (* Byte "n+1 *)
	bZone3RepeatUpDnEnable : BOOL; (* Byte "n+2 *)
	bZone4RepeatUpDnEnable : BOOL; (* Byte "n+3 *)

	iLdGroupNo : INT;
	iUldGroupNo : INT;

	sReservedBool : STRING(95); (* Byte "n+4 ~ n+99" *)

	ARiCallArmNo : ARRAY [0..iProductRecipeStepArrayQty] OF INT; (* Byte "n+100~n+161" *)

	ARiPickStationNo : ARRAY [0..iProductRecipeStepArrayQty] OF INT; (* Byte "n+162~n+223" *)
	ARiTransferStationNo : ARRAY [0..iProductRecipeStepArrayQty] OF INT; (* Byte "n+224~n+285" *)

	ARiDownPickPatternNo : ARRAY [0..iProductRecipeStepArrayQty] OF INT; (* Byte "n+286~n+347" *)
	ARiUpPickPatternNo : ARRAY [0..iProductRecipeStepArrayQty] OF INT; (* Byte "n+348~n+409" *)
	ARiDownTransferPatternNo : ARRAY [0..iProductRecipeStepArrayQty] OF INT; (* Byte "n+410~n+471" *)
	ARiUpTransferPatternNo : ARRAY [0..iProductRecipeStepArrayQty] OF INT; (* Byte "n+472~n+533" *)

	ARiRepeatUpDownCycle : ARRAY [0..iProductRecipeStepArrayQty] OF INT; (* Byte "n+534~n+595" *)

	ARiStnSeqRepNo : ARRAY [0..iProductRecipeStepArrayQty] OF INT; (* Byte "n+596~n+657" *)

	sReservedInt : STRING(41); (* Byte "n+658~n+699" *)

	sDescription : STRING(50); (* Byte "n+700 ~ n+799" *)
	
	bArmRotaryBarrelEnable	: BOOL;


END_STRUCT
END_TYPE

// ---- DUTs/DS TBD/DSV2_ApolloRemoteHoistInput.TcDUT
TYPE DSV2_ApolloRemoteHoistInput :
STRUCT


(*

	iStnQty 									: INT := 12;						(* To change the Qty of Array*)
	iArmQty 									: INT := 2; 						(* ArmQty must lesser than StnQty*)
	iArmSlowPullQty							: INT := 1;
*)

	bPB_EmergencyStop									: BOOL;

	bPB_SelectionSwtich_RemoteEn						: BOOL;
	bPB_SelectionSwtich_JogEn							: BOOL;


	bPB_1stSpd_ArmUp									: BOOL;
	bPB_1stSpd_ArmDown								: BOOL;
	bPB_1stSpd_ArmLeft									: BOOL;
	bPB_1stSpd_ArmRight									: BOOL;
	bPB_1stSpd_ArmHook									: BOOL;
	bPB_1stSpd_ArmUnhook								: BOOL;
	bPB_1stSpd_SlidingDoorOpen							: BOOL;
	bPB_1stSpd_SlidingDoorClose							: BOOL;
	bPB_1stSpd_SlidingDoorClamp							: BOOL;
	bPB_1stSpd_SlidingDoorUnclamp						: BOOL;


	bPB_2ndSpd_ArmUp									: BOOL;
	bPB_2ndSpd_ArmDown								: BOOL;
	bPB_2ndSpd_ArmLeft									: BOOL;
	bPB_2ndSpd_ArmRight								: BOOL;
	bPB_2ndSpd_ArmHook								: BOOL;
	bPB_2ndSpd_ArmUnhook								: BOOL;
	bPB_2ndSpd_SlidingDoorOpen							: BOOL;
	bPB_2ndSpd_SlidingDoorClose							: BOOL;
	bPB_2ndSpd_SlidingDoorClamp						: BOOL;
	bPB_2ndSpd_SlidingDoorUnclamp						: BOOL;



END_STRUCT
END_TYPE

// ---- DUTs/DS TBD/DSV2_ApolloRemoteHoistOutput.TcDUT
TYPE DSV2_ApolloRemoteHoistOutput :
STRUCT


	bArmJogUp										: BOOL;
	bArmJogDown									: BOOL;
	bArmJogLeft										: BOOL;
	bArmJogRight									: BOOL;

	bArmJogVert1stSpeedEn							: BOOL;
	bArmJogVert2ndSpeedEn							: BOOL;

	bArmJogHorz1stSpeedEn							: BOOL;
	bArmJogHorz2ndSpeedEn							: BOOL;

	ARbArmLdVertTopPos								: ARRAY [0..iLdStnQty] OF BOOL;
	ARbArmLdVertBottomPos							: ARRAY [0..iLdStnQty] OF BOOL;
	ARbArmLdHorzHookPos							: ARRAY [0..iLdStnQty] OF BOOL;
	ARbArmLdHorzUnhookPos							: ARRAY [0..iLdStnQty] OF BOOL;

	ARbArmStnVertTopPos							: ARRAY [0..iStnQty] OF BOOL;
	ARbArmStnVertBottomPos							: ARRAY [0..iStnQty] OF BOOL;
	ARbArmStnHorzHookPos							: ARRAY [0..iStnQty] OF BOOL;
	ARbArmStnHorzUnhookPos						: ARRAY [0..iStnQty] OF BOOL;

	ARbArmUldVertTopPos							: ARRAY [0..iUldStnQty] OF BOOL;
	ARbArmUldVertBottomPos							: ARRAY [0..iUldStnQty] OF BOOL;
	ARbArmUldHorzHookPos							: ARRAY [0..iUldStnQty] OF BOOL;
	ARbArmUldHorzUnhookPos						: ARRAY [0..iUldStnQty] OF BOOL;

	ARbStnSlidingDoorOpen							: ARRAY [0..iStnQty] OF BOOL;
	ARbStnSlidingDoorClose							: ARRAY [0..iStnQty] OF BOOL;
	ARbStnSlidingDoorClamp							: ARRAY [0..iStnQty] OF BOOL;
	ARbStnSlidingDoorUnclamp						: ARRAY [0..iStnQty] OF BOOL;

END_STRUCT
END_TYPE

// ---- DUTs/DS TBD/DSV2_ArmPosition.TcDUT
TYPE DSV2_ArmPosition :
STRUCT

	AR3sbTargetPosSt : ARRAY [0..3, 0..iStnQty, 0..12] OF BOOL;
	AR3sbPositionCfm : ARRAY [0..3, 0..iStnQty, 0..12] OF BOOL;
	AR3sb2ndSpdEn : ARRAY [0..3, 0..iStnQty, 0..12] OF BOOL;

	AR3slrPosition : ARRAY [0..3, 0..iStnQty, 0..20] OF LREAL;

(*
	lr2ndSpdRange : LREAL;
	lrPosCfmTolerance : LREAL;
*)

(*Array Declaration -->

Stage 1 --> (0..3) 
------------------------
1=Stn
2=Loading
3=Unloading


Stage 2 --> (0..iStnQty) 
------------------------
No = Station No (Example: 8 = Station 8)



Stage 3 --> (0..12) 
------------------------
1=Vert - Up
2=Vert - SlowPull / Slanted
3=Vert - Regular / Mid Top
4=Vert - AgiUp
5=Vert - AgiDown
6=Vert - Down
7=Horz - Unhook 
8=Horz -  Hook
9=Horz -  Slanted Left
10=Horz - Slanted Right
11=Lifter - Up 
12=Lifter - down 
13=Reserved
14=Reserved
15=Reserved
16=Reserved
17=Reserved
18=Reserved
19=Reserved
20=Reserved

*)

END_STRUCT
END_TYPE

// ---- DUTs/DS TBD/DSV2_BasketInfo.TcDUT
TYPE DSV2_BasketInfo : (*Full Occupied Byte = 700*)

(*[][][][][][][][][][]----- Basket Information - Attached with Basket -----[][][][][][][][][][]*)

STRUCT
	bAvailibility : BOOL; (* Byte "n" *)
	bAvailibility_A : BOOL; (* Byte "n" *)
	bAvailibility_B : BOOL; (* Byte "n" *)
	sReservedBool : STRING(97); (* Byte "n+2~n+99" *)

	iProductRecipeNo : INT; (* Byte "n+100, n+101" *)
	iProductRecipeStepNo : INT; (* Byte "n+102, n+103" *)
	iStationSeqenceRecipeNo : INT; (* Byte "n+104, n+105" *)
	iPreviousStationNo : INT; (* Byte "n+106, n+107" *)
	iCurrentStationNo : INT; (* Byte "n+108, n+109" *)
	sReservedInt : STRING(87); (* Byte "n+112~n+199" *)


	sProgramDescription : STRING(50) ; (* Byte "n+200~n+299" *)
	sProductID : STRING(50); (* Byte "n+300~n+399" *)
	ARsBarcodeData : ARRAY [0..10] OF STRING(50); (* Byte "n+400~n+499" *)
	sFilePath : STRING(50); (* Byte "n+500~n+599" *)
	sProductQuality : STRING(50); (* Byte "n+600~n+699" *)

	DSV2MinMaxEffTime : DSV2_MinMaxEffTime;

(*
	sBarcodeData Information
	[0] - No in use 
	[1] - Barcode for Program No (DEFAULT)	
	[2] - Barcode for Logging
	[3] - Barcode for Logging
	[4] - Barcode for Logging
	[5] - Barcode for Logging
	[6] - Barcode for Logging
	[7] - Barcode for Logging
	[8] - Barcode for Logging
	[9] - Barcode for Logging
	[10] - Barcode for Logging
*)


END_STRUCT
END_TYPE

// ---- DUTs/DS TBD/DSV2_ClangsonicGenerator.TcDUT
TYPE DSV2_ClangsonicGenerator :
STRUCT

	iRWRef 						: ARRAY [1..iUSModbusRWQty] OF INT;
	(***************************************************)
	(*
		0 = --- End Code ---
		1 = Read ONLY
		2 = Read/Write
		3 = Disable
		4 = --- End Code ---
		Above 4 = --- End Code ---
										*)
	(***************************************************)

	wModbusData 				: ARRAY [1..iUSModbusRWQty] OF WORD; (*Data for Read or Write*)
	wModbusRegisterAddr 		: ARRAY [1..iUSModbusRWQty] OF WORD; (*Modbus Register Address*)
	B_UnitID 						: ARRAY [1..iUSModbusRWQty] OF BYTE; (*Unit ID - Modbus ID*)

END_STRUCT
END_TYPE

// ---- DUTs/DS TBD/DSV2_fbGnrProductRecipeMemoryOut.TcDUT
TYPE DSV2_fbGnrProductRecipeMemoryOut : (*Full Occupied Byte = 1700*)
STRUCT

	bCallCompleted 							: BOOL; (* Byte "n" *)

	bInvalidProductRecipeNoErrHold 		: BOOL; (* Byte "n+1" *)
	bInvalidProductRecipeNoErrPulse		: BOOL; (* Byte "n+2" *)
	bInvalidProductRecipeStepErrHold 		: BOOL; (* Byte "n+3" *)
	bInvalidProductRecipeStepErrPulse		: BOOL; (* Byte "n+4" *)

	bCallUpDownPatternMemoryErr 			: BOOL; (* Byte "n+5" *)
	bCallArmSpeedProfileMemoryErr 		: BOOL; (* Byte "n+6" *)
	bCallPickStationNoErr 					: BOOL; (* Byte "n+7" *)
	bCallTransferStationNoErr 				: BOOL; (* Byte "n+8" *)

	sReservedBool 							: STRING(90); (* Byte "n+9~n+99" *)


	iCalledProductRecipeNo 					: INT; (* Byte "n+100~n+101" *) (*New*)
	iCalledProductRecipeStep				: INT; (* Byte "n+102~n+103" *) (*New*)
	iCallCaseNo 								: INT; (* Byte "n+104~n+105" *)

	sReservedInt 								: STRING(93); (* Byte "n+106~n+199" *)

	sProductRecipeDescription 				: STRING(50);

	DSGnrCalledArmPnpParameter : DSV2_Gnr_CalledArmPnpParameter;

END_STRUCT
END_TYPE

// ---- DUTs/DS TBD/DSV2_fbStationSequenceRecipeCall.TcDUT
TYPE DSV2_fbStationSequenceRecipeCall : (*Full Occupied Byte = 500*)
STRUCT
	bCallPB: BOOL; (* Byte "n" *)
	bCallCompleted : BOOL; (* Byte "n+1" *)
	bInvalidCallStationSequenceNoHold : BOOL; (* Byte "n+2" *)
	bInvalidCallStationSequenceNoPulse : BOOL; (* Byte "n+3" *)
	sReservedBool : STRING(95); (* Byte "n+4~n+99" *)


	Call_iStationSequenceRecipe : INT; (* Byte "n+100, n+101" *)
	sReservedInt : STRING(97); (* Byte "n+102~n+199" *)


	Call_sSequenceRecipeDescription : STRING(50); (* Byte "n+200~n+299" *)


	Call_DsStationSequenceRecipeMemory : DSV2_StationSequenceRecipeMemory; (* Byte "n+300 onward" *)





END_STRUCT
END_TYPE

// ---- DUTs/DS TBD/DSV2_fbStationSequenceRecipeStore.TcDUT
TYPE DSV2_fbStationSequenceRecipeStore : (*Full Occupied Byte = 500*)
STRUCT

	bCopyPB : BOOL; (* Byte "n" *)
	sReservedBool : STRING(98); (* Byte "n+1~n+99" *)


	iStationSequenceRecipeNo: INT; (* Byte "n+100, n+101" *)	(* 10 sets of Station Sequence Recipe *)
	iCopyToSubRecipeNo : INT; (* Byte "n+102, n+103" *)
	sReservedInt : STRING(95); (* Byte "n+104~n+199" *)


	sStationSequenceRecipeDescription : STRING(50); (* Byte "n+200~n+299" *)  (* Description of Station Sequence Recipe - Naming*)


	DsStationSequenceRecipeMemory : DSV2_StationSequenceRecipeMemory; (* Byte "n+300 onward" *)






END_STRUCT
END_TYPE

// ---- DUTs/DS TBD/DSV2_Gnr_CalledArmPnpParameter.TcDUT
TYPE DSV2_Gnr_CalledArmPnpParameter : (*Full Occupied Byte = 1400*)
STRUCT

	iCallArmNo : INT; (* Byte "n~, n+1" *)
	iStnSeqRecipeNo : INT; (* Byte "n+2, n+3" *)
	iPickStationNo : INT; (* Byte "n+4, n+5" *)
	iTransferStationNo : INT; (* Byte "n+6, n+7" *)

	iLdGroupNo : INT;
	iUldGroupNo : INT;

	iDrippingTimeSV : INT; (* Byte "n+8, n+9" *)

	sReservedInt : STRING(189); (* Byte "n+10~n+199" *)

	DSA1DownPickMovement : DSA1_UpDownMovement;
	DSA1UpPickMovement : DSA1_UpDownMovement;
	DSA1DownTransferMovement : DSA1_UpDownMovement;
	DSA1UpTransferMovement : DSA1_UpDownMovement;

END_STRUCT
END_TYPE

// ---- DUTs/DS TBD/DSV2_MinMaxEffTime.TcDUT
TYPE DSV2_MinMaxEffTime :
STRUCT
	iProductRecipeNo			: INT;
	ARiTransferStationNo		: ARRAY [0..iProductRecipeStepArrayQty] OF INT;
	ARiStnSeqRepNo 		: ARRAY [0..iProductRecipeStepArrayQty] OF INT;
	ARiMinTime 				: ARRAY [0..iProductRecipeStepArrayQty] OF INT;
	ARiMaxTime 				: ARRAY [0..iProductRecipeStepArrayQty] OF INT;
	ARiEffTime 				: ARRAY [0..iProductRecipeStepArrayQty] OF INT;

END_STRUCT
END_TYPE

// ---- DUTs/DS TBD/DSV2_ModbusControl.TcDUT
TYPE DSV2_ModbusControl :
STRUCT

	iRWRef 						: ARRAY [1..iModbusRWQty] OF INT;
	(***************************************************)
	(*
		0 = --- End Code ---
		1 = Read ONLY
		2 = Read/Write
		3 = Disable
		4 = --- End Code ---
		Above 4 = --- End Code ---
										*)
	(***************************************************)

	wModbusData 				: ARRAY [1..iModbusRWQty] OF WORD; (*Data for Read or Write*)
	wModbusRegisterAddr 		: ARRAY [1..iModbusRWQty] OF WORD; (*Modbus Register Address*)
	B_UnitID 						: ARRAY [1..iModbusRWQty] OF BYTE; (*Unit ID - Modbus ID*)

END_STRUCT
END_TYPE

// ---- DUTs/DS TBD/DSV2_SSERSourceMinMaxTime.TcDUT
TYPE DSV2_SSERSourceMinMaxTime :
STRUCT

	ARiMinTime : ARRAY [0..iStationSequenceRecipeArrayQty] OF INT;
	ARiMaxTime : ARRAY [0..iStationSequenceRecipeArrayQty] OF INT;
	ARiEffTime : ARRAY [0..iStationSequenceRecipeArrayQty] OF INT;

END_STRUCT
END_TYPE

// ---- DUTs/DS TBD/DSV2_StationSequenceRecipeMemory.TcDUT
TYPE DSV2_StationSequenceRecipeMemory : (*Full Occupied Byte = 200*)
STRUCT

	sReservedBool 				: STRING(50); (* Byte "n+0 ~ n+99" *)

	AR10iStationSubProNo 		: ARRAY [0..iProductRecipeStepArrayQty] OF INT; (* Byte "n100~n+121" *) (* 10 units of SubProcessProgramNo / Steps *)
	AR10iCycle 					: ARRAY [0..iProductRecipeStepArrayQty] OF INT; (* Byte "n+122~n+143" *) (* 10 units of Integer to Store the Cycle needed on the specified Steps. at least "1" *)
	AR10iRepeatFromStepNo 	: ARRAY [0..iProductRecipeStepArrayQty] OF INT; (* Byte "n+144~n+165" *) (* 10 units of Integer to when Cycle repeat, it will repeat from Which Steps  *)
	sReservedInt 					: STRING(33); (* Byte "n+166~n+199" *)

(*Added*)
	iProcessMinTime				: INT;
	iProcessMaxTime				: INT;

	iProcessCalculatedTime		: INT;

(*Added by LEE - SSER Min Time and Cycle Auto Calculated*)
	iCycleProcessTime			: INT;
	iCycleCalculated				: INT;
	iCycleRemainingTime			: INT;
	iStepOverwriteCycle			: INT;



END_STRUCT
END_TYPE

// ---- DUTs/DS TBD/DSV2_StnMinMaxEffTIme.TcDUT
TYPE DSV2_StnMinMaxEffTIme :
STRUCT
	iMinTime 				: INT;
	iMaxTime 				: INT;
	iEffTime 					: INT;

END_STRUCT
END_TYPE

// ---- DUTs/DS TBD/DSV2_TimeTrackerInput.TcDUT
TYPE DSV2_TimeTrackerInput :
STRUCT
(* from DSA1_PnpSequenceMemory*)

(*	bTimeTrackerEn : BOOL;*)
	iTimeTrackerProductRecipeNo : INT;
(*	iTimeTrackerStepNo : INT; (*Byte "n+110, n+111" *) (***************NEW******************)*)

	iLdGroupNo : INT;
	iUldGroupNo : INT;

	ARiCallArmNo : ARRAY [0..iProductRecipeStepArrayQty] OF INT; (* Byte "n+100~n+161" *)

	ARiPickStationNo : ARRAY [0..iProductRecipeStepArrayQty] OF INT; (* Byte "n+162~n+223" *)
	ARiTransferStationNo : ARRAY [0..iProductRecipeStepArrayQty] OF INT; (* Byte "n+224~n+285" *)

	ARiStnSeqRepNo : ARRAY [0..iProductRecipeStepArrayQty] OF INT; (* Byte "n+596~n+657" *)

END_STRUCT

END_TYPE

// ---- DUTs/DS TBD/DSV3_BarcodeRegistration.TcDUT
TYPE DSV3_BarcodeRegistration :
STRUCT

	sBarcodeRegistered															 : STRING(99);
	iLinkProductRecipeNo															 : INT;
	bBarcodeRegistrationEn 														 : BOOL;
	sLinkProductRecipeDescription													 : STRING(99);

END_STRUCT
END_TYPE

// ---- DUTs/DS TBD/DSV3_JRS_Alarm.TcDUT
TYPE DSV3_JRS_Alarm :
STRUCT
	b200_00_FreshHCTankCircPumpTORAlarm					: BOOL;
	b200_01_CircTankCircPumpTORAlarm 						: BOOL;
	b200_02_ThermalOilPumpTORAlarm							: BOOL;
	b200_03_ThermalOilLowLevelAlarm 							: BOOL;
	b200_04_ThermalOilTempHighAlarm 						: BOOL;
	b200_05_ThermalOilTempNotReadyAlarm 					: BOOL;
	b200_06_ThermalOilHeaterOnOffAlarm 						: BOOL;
	b200_07_TopDistillatorTempHighAlarm					 	: BOOL;
	b200_08_TopDistillatorTempNotReadyAlarm 					: BOOL;
	b200_09_TopDistillatorHeaterOnOffAlarm 						: BOOL;
	b200_10_RecycleStartStopPBAlarm 							: BOOL;
	b200_11_EstopPBAlarm 									: BOOL;

	b201_00_PhaseSeqenceRelayAlarm 						: BOOL;
	b201_01_ThermalOilUpThermostatAlarm 						: BOOL;
	b201_02_SludgeTankHighLevelAlarm 						: BOOL;
	b201_03_FreshHCTankLowLevelAlarm 						: BOOL;
	b201_04_VacuumNotAchieveAlarm 							: BOOL;
	b201_05_IncomingCDALowPressureAlarm 					: BOOL;
	b201_06_CoolingWaterLowFlowAlarm 						: BOOL;
	b201_07_CircularTankLowLevelAlarm 						: BOOL;
	b201_08_BottomDistillatorTempHighAlarm 					: BOOL;
	b201_09_BottomDistillatorTempNotReadyAlarm				: BOOL;
	b201_10_BottomDistillatorHeaterOnOffAlarm					: BOOL;
	b201_11_ThermalOilDownThermostatAlarm 					: BOOL;
	b201_12_ThermalOilMidThermostatAlarm 						: BOOL; (*New Added- Lee, 190109*)

	b202_00_VaporGenerationTempHighAlarm 					: BOOL;
	b202_01_VaporGenerationTempNotReadyAlarm 				: BOOL;
	b202_02_VaporGenerationHeaterOnOffAlarm 					: BOOL;
	b202_03_WasteCollectionTankLowLevelAlarm 				: BOOL;
	b202_04_VaporGenerationTankLowLevelAlarm 				: BOOL;
	b202_05_HCPurgingAV3_1Alarm 							: BOOL;
	b202_06_MainMachineWasteTankLowLevelAlarm 				: BOOL;
	b202_07_MainMachineWasteTankHighLevelAlarm 				: BOOL;
	b202_08_ReservedAlarm 									: BOOL;
	b202_09_ReservedAlarm 									: BOOL;
	b202_10_ReservedAlarm 									: BOOL;
	b202_11_ReservedAlarm 									: BOOL;

	b203_00_ChillerSelectorOnOffAlarm 							: BOOL;
	b203_01_ColdWaterTankLowLevelAlarm 						: BOOL;
	b203_02_SludgeTankMissingAlarm 							: BOOL;
	b203_03_ColdWaterTankTempHighAlarm 					: BOOL;
	b203_04_ColdWaterTankTempNotReadyAlarm 				: BOOL;
	b203_05_ColdWaterTankHeaterOnOffAlarm 					: BOOL;
	b203_06_ChillerPumpTORAlarm 							: BOOL;
	b203_07_ChillerFlowSwitchAlarm 							: BOOL;
	b203_08_ChillerInterlockRelayAlarm 							: BOOL;
	b203_09_ReservedAlarm 									: BOOL;
	b203_10_ThermalOilChangeWarning 							: BOOL;
	b203_11_ThermalOilChangeAlarm 							: BOOL;


END_STRUCT
END_TYPE

// ---- DUTs/DS TBD/DSV3_JRS_HMI.TcDUT
TYPE DSV3_JRS_HMI :
STRUCT


	bTarget_JRSZeroVacuumLvlSavePB 					: BOOL;
	bTarget_JRSHighVacuumLvlSavePB 					: BOOL;
	lrTarget_JRSHighVacuumRefReading 					: LREAL;
	rTarget_JRSVacuumLevelPV_kPa 						: REAL;
	rTarget_JRSVacuumLevelSV_kPa 						: REAL;

	rTarget_ThermalOilTempPV 							: REAL;
	rTarget_ThermalOilTempHighAlarmSV 					: REAL;
	rTarget_ThermalOilTempReadySV 						: REAL;
	rTarget_ThermalOilTempOnOffSV 						: REAL;
	rTarget_ThermalOilTempOnOffHysSV 					: REAL;
	rTarget_ThermalOilAnalogInputFineTuneRatio				: REAL;

	rTarget_TopDistillatorTempPV 							: REAL;
	rTarget_TopDistillatorTempHighAlarmSV 					: REAL;
	rTarget_TopDistillatorTempReadySV 					: REAL;
	rTarget_TopDistillatorTempOnOffSV 						: REAL;
	rTarget_TopDistillatorTempOnOffHysSV 					: REAL;
	rTarget_TopDistillatorAnalogInputFineTuneRatio			: REAL;

	rTarget_BottomDistillatorTempPV 						: REAL;
	rTarget_BottomDistillatorTempHighAlarmSV 				: REAL;
	rTarget_BottomDistillatorTempReadySV 					: REAL;
	rTarget_BottomDistillatorTempOnOffSV 					: REAL;
	rTarget_BottomDistillatorTempOnOffHysSV 				: REAL;
	rTarget_BottomDistillatorAnalogInputFineTuneRatio		: REAL;

	rTarget_VaporGenerationTempPV 						: REAL;
	rTarget_VaporGenerationTempHighAlarmSV 				: REAL;
	rTarget_VaporGenerationTempReadySV 				: REAL;
	rTarget_VaporGenerationTempOnOffSV 					: REAL;
	rTarget_VaporGenerationTempOnOffHysSV 				: REAL;
	rTarget_VaporGenerationAnalogInputFineTuneRatio		: REAL;

	rTarget_ColdWaterTankTempPV 						: REAL;
	rTarget_ColdWaterTankTempHighAlarmSV 				: REAL;
	rTarget_ColdWaterTankTempReadySV 					: REAL;
	rTarget_ColdWaterTankTempOnOffSV 					: REAL;
	rTarget_ColdWaterTankTempOnOffHysSV 				: REAL;
	rTarget_ColdWaterAnalogInputFineTuneRatio				: REAL;

	b1000_00_AutoModeOnOffPB 							: BOOL;
	b1000_01_AutoOriginOnOffPB 							: BOOL;
	b1000_02_AutoPreparationOnOffPB 						: BOOL;
	b1000_03_AutoModeStartStopPB 						: BOOL;
	b1000_04_Reserved 									: BOOL;
	b1000_05_AutoCycleStopPB 							: BOOL;
	b1000_06_AutoBoilingStart 								: BOOL;
	b1000_07_AutoBoilingDownCompletedFlag 				: BOOL;
	b1000_08_AutoBoilingSludgeDrainCompletedFlag 			: BOOL;
	b1000_09_AutoBoilingDistrillatorDrainCompletedFlag 		: BOOL;
	b1000_10_Reserved 									: BOOL;
	b1000_11_Reserved 									: BOOL;
	b1000_12_Reserved 									: BOOL;
	b1000_13_AutoProgressStopRE 						: BOOL;
	b1000_14_AlarmResetPB 								: BOOL;
	b1000_15_BuzzerResetPB 								: BOOL;

	b9000_09_AutoBoilSludgeDrainCoolingCompletedFlag 		: BOOL;    (************* New extra request by customer - YCH************)
	b9000_15_AutoBoilingCompletedFlag 					: BOOL;    (************* New extra request by customer - YCH************)

	b1001_01_AutoOriginCompletedFlag 						: BOOL;
	b1001_02_AutoPreparationCompletedFlag 				: BOOL;
	b1001_03_Reserved 									: BOOL;
	b1001_04_Reserved 									: BOOL;
	b1001_05_Reserved 									: BOOL;
	b1001_06_ManualBoilingPageInRangeFlag 				: BOOL;
	b1001_07_Reserved 									: BOOL;
	b1001_08_Reserved 									: BOOL;
	b1001_09_ManualPageInRangeFlag 						: BOOL;
	b1001_10_AutoProgressFlag 							: BOOL;
	b1001_11_Reserved 									: BOOL;
	b1001_12_Reserved 									: BOOL;
	b1001_13_Reserved 									: BOOL;
	b1001_14_EmergencyStopAlarm 						: BOOL;
	b1001_15_AlarmOccur 									: BOOL;

	b1020_00_ManualBoilingCycleCompleteFlag 				: BOOL;

	b1030_00_ManualBoilingStartStopPB 					: BOOL;
	b1030_01_ManualBoilingProgressHR 					: BOOL;
	b1030_02_ManualBoilDownCompletedFlag 				: BOOL;
	b1030_03_ManualBoilSludgeCoolingCompletedFlag 		: BOOL;
	b1030_04_ManualBoilSludgeDrainCompletedFlag 			: BOOL;
	b1030_05_Reserved 									: BOOL;
	b1030_06_ChillerOn 									: BOOL;
	b1030_07_ManualChillerOn 								: BOOL;
	b1030_08_ManualBoilingStop 							: BOOL;
	b1030_09_ManualBoilingStartHR 						: BOOL;
	b1030_10_Reserved 									: BOOL;
	b1030_11_Reserved 									: BOOL;
	b1030_12_Reserved 									: BOOL;
	b1030_13_Reserved 									: BOOL;
	b1030_14_Reserved 									: BOOL;
	b1030_15_ManualBoilingStartStopPB 					: BOOL;

	b1040_00_ThermalOilChangeHMeterAlarm 				: BOOL;
	b1040_01_ThermalOilChangeHMeterResetPB 				: BOOL;
	b1040_02_ThermalOiChangeWarning 					: BOOL;

	b1200_00_VaporRequestStartHR 						: BOOL;
	b1200_01_VaporRequestStopHR 						: BOOL;

	bH130_00_AutoBoilingModeOff 							: BOOL; (*Add New*)
	b1300_00_ManualBoilDownStartMode 					: BOOL;
	b1300_01_ManualBoilingDownStartPBTS 					: BOOL;

	bRecycleStartStopPB									: BOOL;
	bChillerSelectorOnOff									: BOOL;

	iD0_HMICurrentPage 									: INT;

	sD100_MessageDisplay 								: STRING;
	iD100_MessageDisplay 								: INT;
	iD200_AutoBoilProcessTimeSV_Min 						: INT;
	iD201_AutoBoilDownTimeSV_Min 						: INT;
	iD202_AutoBoilDistillatorDrainTimeSV_Sec 				: INT;
	iD203_AutoBoilSludgeDrainTimeSV_Sec 					: INT;
(*	iD204_60SecDelayTime 								: INT;*)
	iD205_5SecDelayTime 								: INT;

	iD890_AutoBoilSludgeDrainCoolingProcessTimeSV_Min 	: INT;    (************* New extra request by customer - YCH************)

	iD210_ManualBoilDownTimeSV_Min 						: INT;
	iD211_ManualBoilSludgeCoolingTimeSV_Min 				: INT;
	iD212_ManualBoilSludgeDrainSV_Sec 					: INT;

	iD220_AutoBoilProcessTimePV_Min 						: INT;
	iD225_AutoBoilProcessTimePV_Sec 					: INT;

	iD221_AutoBoilDownTimePV_Min 						: INT;
	iD226_AutoBoilDownTimePV_Sec 						: INT;

	iD222_AutoBoilDistillatorDrainTimePV_Sec 				: INT;
	iD223_AutoBoilSludgeDrainTimePV_Sec 					: INT;

	iD990_AutoBoilSludgeDrainCoolingProcessTimePV_Min 	: INT;    (************* New extra request by customer - YCH************)
	iD991_AutoBoilSludgeDrainCoolingProcessTimePV_Sec 	: INT;    (************* New extra request by customer - YCH************)

	iD230_ManualBoilDownTimePV_Min 						: INT;
	iD231_ManualBoilSludgeCoolingTimePV_Min 				: INT;
	iD232_ManualBoilSludgeDrainPV_Sec 					: INT;

	iD235_ManualBoilDownTimePV_Sec 					: INT;
	iD236_ManualBoilSludgeCoolingTimePV_Sec 			: INT;

	iD240_ThermalOilChangeHMeterPV_Hour 				: INT;
	iD241_ThermalOilChangeHMeterPV_Min 					: INT;
	iD242_ThermalOilChangeHMeterPV_Sec 					: INT;

	iD250_ThermalOilChangeWarningSV_Hour 				: INT;
	iD251_ThermalOilChangeAlarmSV_Hour 					: INT;

	iD300_AutoModeTimeValue 							: INT;

	iD400_0SecDelayAlarm 								: INT;
	iD401_3SecDelayAlarm 								: INT;
	iD402_10SecDelayAlarm 								: INT;
	iD403_30SecDelayAlarm 								: INT;
	iD404_60SecDelayAlarm 								: INT;
	iD405_5SecDelayAlarm 								: INT;

	iD480_ManualBoilingDrainCyclePV 						: INT;

	iD490_ManualBoilCycleSV 								: INT;

	iJRS_AlarmDaysSV_Routine							: INT ;
         iJRS_AlarmDaysSV_Major							         : INT ;
         iJRS_WarningDaysSV_Routine						         : INT ;
	iJRS_WarningDaysSV_Major							: INT ;
	iJRS_RunDaysPV_Routine								: INT;
 	iJRS_RunDaysPV_Major								: INT;

	bJRS_ServiceAlarm_Routine							: BOOL;
	bJRS_ServiceAlarm_Major							     	: BOOL;
	bJRS_ServiceWarning_Routine							: BOOL;
	bJRS_ServiceWarning_Major							: BOOL;

	bJRS_DaysPvReset_Routine							: BOOL;
	bJRS_DaysPvReset_Major								: BOOL;
	sJRS_PreviousDateJRS_Routine						: STRING ;
	sJRS_PreviousDateJRS_Major							: STRING ;

 	sJRS_CurrentDate										: STRING;
	bPowerDelay											: BOOL;

END_STRUCT


END_TYPE

// ---- DUTs/DS TBD/DSV3_JRS_Input.TcDUT
TYPE DSV3_JRS_Input :

STRUCT

(*Channel 0*)
	b000_00_FreshHCTankCircPumpTOR 											: BOOL;
	b000_01_CircTankCircPumpTOR 												: BOOL;
	b000_02_ThermalOilPumpTOR													: BOOL;
	b000_03_ThermalOilLevelSensor												: BOOL;
	b000_04_ThermalOilTempCtrlHighTempAlarmSignal								: BOOL;
	b000_05_ThermalOilTempCtrlReadySignal										: BOOL;
	b000_06_ThermalOilTempCtrlOnOffSignal 										: BOOL;
	b000_07_TopDistillatorTempCtrlHighTempAlarmSignal								: BOOL;
	b000_08_TopDistillatorTempCtrlReadySignal										: BOOL;
	b000_09_TopDistillatorTempCtrlOnOffSignal 										: BOOL;
	b000_10_RecycleStartStopPB			 										: BOOL;
	b000_11_EStopPB															: BOOL;

(*Channel 1*)
	b001_00_PhaseSequenceRelayAlarm											: BOOL;
	b001_01_ThermalOilUpThermostat 												: BOOL;
	b001_02_SludgeTankLevelSensor												: BOOL;
	b001_03_FreshHCTankLevelSensor												: BOOL;
	b001_04_VacuumNotAchieveSignal												: BOOL;
	b001_05_IncomingCDAPressureSwitch											: BOOL;
	b001_06_CoolingWaterFlowSwitch	 											: BOOL;
	b001_07_CircularTankLevelSensor												: BOOL;
	b001_08_BottomDistillatorTempCtrlHighTempAlarmSignal							: BOOL;
	b001_09_BottomDistillatorTempCtrlReadySignal									: BOOL;
	b001_10_BottomDistillatorTempCtrlOnOffSignal 									: BOOL;
	b001_11_ThermalOilDownThermostat											: BOOL;
	b001_12_ThermalOilMidThermostat												: BOOL; (*New Added- Lee, 190109*)

(*Channel 2*)
	b002_00_VaporGenerationTempCtrlHighTempAlarmSignal							: BOOL;
	b002_01_VaporGenerationTempCtrlReadySignal									: BOOL;
	b002_02_VaporGenerationTempCtrlOnOffSignal									: BOOL;
	b002_03_WasteCollectionTankLevelSensor										: BOOL;
	b002_04_VaporGenerationTankLowLevelSensor									: BOOL;
	b002_05_HCPurgingAV														: BOOL;
	b002_06_MainMachineWasteCollectTankLowLevelSignal							: BOOL;
	b002_07_MainMachineWasteCollectTankHighLevelSignal							: BOOL;
	b002_08_FromMainMachineSignal3												: BOOL;
	b002_09_FromMainMachineSignal4												: BOOL;
	b002_10_FromMainMachineSignal5												: BOOL;
	b002_11_ReservedAlarmSignal													: BOOL;

(*Channel 3*)
	b003_00_ChillerSelectorOnOff													: BOOL;
	b003_01_ColdWaterTankLowLevelSensor										: BOOL;
	b003_02_SludgeTankPresentSensor												: BOOL;
	b003_03_ColdWaterTankTempCtrlHighTempAlarmSignal							: BOOL;
	b003_04_ColdWaterTankTempCtrlReadySignal									: BOOL;
	b003_05_ColdWaterTankTempCtrlOnOffSignal										: BOOL;
	b003_06_ChillerPumpTOR														: BOOL;
	b003_07_ChillerFlowSwitch														: BOOL;
	b003_08_ChillerInterlockRelay													: BOOL;
	b003_09_ReservedAlarmSignal													: BOOL;
	b003_10_ReservedAlarmSignal													: BOOL;
	b003_11_ReservedAlarmSignal													: BOOL;


END_STRUCT
END_TYPE

// ---- DUTs/DS TBD/DSV3_JRS_Output.TcDUT
TYPE DSV3_JRS_Output :
STRUCT

(*Channel 100*)
	b100_00_FreshHCTankCircPumpOnOff 											: BOOL;
	b100_01_CircTankCircPumpOnOff												: BOOL;
	b100_02_ThermalOilPumpOnOff													: BOOL;
	b100_03_ThermalOilHeaterOnOff												: BOOL;
	b100_04_Buzzer																: BOOL;
	b100_05_RecycleStartStopIndicator												: BOOL;
	b100_06_Reserved															: BOOL;
	b100_07_UFOVacuumRelease32WayAV											: BOOL;

(*Channel 101*)
	b101_00_CondenserTankVacuumReleaseAV										: BOOL;
	b101_01_WasteSludgeCollectionDrumAV 											: BOOL;
	b101_02_DistillationTankDrainAV												: BOOL;
	b101_03_EconomizerAV														: BOOL;
	b101_04_Reserved															: BOOL;
	b101_05_Reserved															: BOOL;
	b101_06_VaporGenerationAV			 										: BOOL;
	b101_07_VacuumSharingAV													: BOOL;

(*Channel 102*)
	b102_00_RecycleReadySignal													: BOOL;
	b102_01_VaporNotAvailableForRequestSignal									: BOOL;
	b102_02_ToMainMachineSignal3												: BOOL;
	b102_03_ToMainMachineSignal4												: BOOL;
	b102_04_ToMainMachineSignal5												: BOOL;
	b102_05_Reserved															: BOOL;
	b102_06_Reserved															: BOOL;
	b102_07_Reserved															: BOOL;

(*Channel 103*)
	b103_00_ChillerPumpOnOff														: BOOL;
	b103_01_Reserved															: BOOL;
	b103_02_Reserved															: BOOL;
	b103_03_Reserved															: BOOL;
	b103_04_ChillerSelectorOnOffIndicator											: BOOL;
	b103_05_ChillerReadySignal													: BOOL;
	b103_06_ChillerCompressorOnOff												: BOOL;
	b103_07_Reserved															: BOOL;



(*Channel 100*)
	i100_00_FreshHCTankCircPumpOnOff 											: INT;
	i100_01_CircTankCircPumpOnOff												: INT;
	i100_02_ThermalOilPumpOnOff													: INT;
	i100_03_ThermalOilHeaterOnOff													: INT;
	i100_04_Buzzer																: INT;
	i100_05_RecycleStartStopIndicator												: INT;
	i100_06_Reserved															: INT;
	i100_07_UFOVacuumRelease32WayAV											: INT;

(*Channel 101*)
	i101_00_CondenserTankVacuumReleaseAV										: INT;
	i101_01_WasteSludgeCollectionDrumAV 											: INT;
	i101_02_DistillationTankDrainAV													: INT;
	i101_03_EconomizerAV														: INT;
	i101_04_Reserved															: INT;
	i101_05_Reserved															: INT;
	i101_06_VaporGenerationAV		 											: INT;
	i101_07_VacuumSharingAV														: INT;

(*Channel 102*)
	i102_00_RecycleReadySignal													: INT;
	i102_01_VaporNotAvailableForRequestSignal										: INT;
	i102_02_ToMainMachineSignal3													: INT;
	i102_03_ToMainMachineSignal4													: INT;
	i102_04_ToMainMachineSignal5													: INT;
	i102_05_Reserved															: INT;
	i102_06_Reserved															: INT;
	i102_07_Reserved															: INT;

(*Channel 103*)
	i103_00_ChillerPumpOnOff														: INT;
	i103_01_Reserved															: INT;
	i103_02_Reserved															: INT;
	i103_03_Reserved															: INT;
	i103_04_ChillerSelectorOnOffIndicator												: INT;
	i103_05_ChillerReadySignal													: INT;
	i103_06_ChillerCompressorOnOff												: INT;
	i103_07_Reserved															: INT;


END_STRUCT
END_TYPE

// ---- DUTs/DS TBD/DSV3_StnInterlock.TcDUT
TYPE DSV3_StnInterlock :
STRUCT

	ARbArmDownInterlock 	: ARRAY [0..iStnQty] OF BOOL;
	ARbArmUpInterlock 		: ARRAY [0..iStnQty] OF BOOL;

END_STRUCT
END_TYPE

// ---- DUTs/DS TBD/DSV3_TempCtrlParameter.TcDUT
TYPE DSV3_TempCtrlParameter :
STRUCT

	rProTankHighTempSV				:  REAL;
	rProTank1stLimitTempSV			:  REAL;
	rProTankProcessTempSV			:  REAL;
	rProTankRdyTempSV				:  REAL;
	rProTankHysTempSV				:  REAL;
	iProTankRdyTempDelayTime		:  INT;

	rSubTankHighTempSV			:  REAL;
	rSubTank1stLimitTempSV			:  REAL;
	rSubTankProcessTempSV			:  REAL;
	rSubTankRdyTempSV				:  REAL;
	rSubTankHysTempSV				:  REAL;
	iSubTankRdyTempDelayTime		:  INT;


END_STRUCT
END_TYPE

// ---- DUTs/DS TBD/DSV3_TempCtrlRecipe.TcDUT
TYPE DSV3_TempCtrlRecipe :
STRUCT
	Station: ARRAY [0..iStnQty] OF DSV3_TempCtrlParameter;

END_STRUCT
END_TYPE

// ---- DUTs/DS TBD/DSV3_XML_Recipe.TcDUT
TYPE DSV3_XML_Recipe :
STRUCT


	DSProductRecipe			 								: DSV2_A1_PnpSequenceMemory;
	AR2SiRecipeTimeBlockNoCallArmTime 						: ARRAY[1..iRecipeBlockQty, 1..9] OF INT;
	AR2SiRecipeTimeBlockWithCallArmTime 					: ARRAY[1..iRecipeBlockQty, 1..9] OF INT;
	bProductRecipeTimeBlockAvailable 							:  BOOL;
	DSTempCtrlRecipe 										:  DSV3_TempCtrlRecipe;


	(*

		PRODUCT RECIPE MEMORY
			Need to read/write to below (Location: B_JKS_NewFB_V2 -> FBP-Memory Sub -> fbV2_A1_PnpSequenceMemory )
			- Declare single memory refer to this Declaration-> ARDsPnpSequenceMemory : ARRAY [1..iProductRecipeArrayQty] OF DSA1_PnpSequenceMemory;



		TRACKER MEMORY (Info)
			Need to declared as below
			AR2SiCalledRecipeTimeBlockNoCallArmTime 			: ARRAY[1..iRecipeBlockQty, 1..9] OF INT;
			AR2SiCalledRecipeTimeBlockWithCallArmTime 			: ARRAY[1..iRecipeBlockQty, 1..9] OF INT;
				
			Need to read/write to below (Location: B_JKS_NewFB_V2 -> FBP_ProcessOptimisation -> fbV2_FBPTimeTrackerG3 )
			AR3SiRecipeTimeBlockMemoryNoCallArmTime						: ARRAY [1..iProductRecipeArrayQty, 1..iRecipeBlockQty, 1..9] OF INT;
			AR3SiRecipeTimeBlockMemoryWithCallArmTime						: ARRAY [1..iProductRecipeArrayQty, 1..iRecipeBlockQty, 1..9] OF INT;


		TRACKER Status (BOOL)
			Need to read/write to below (Location: B_JKS_NewFB_V2 -> FBP_ProcessOptimisation -> fbV2_FBPTimeTrackerG3 )
			ARbProductRecipeTimeBlockAvailable 					: ARRAY [0..iProductRecipeArrayQty] OF BOOL;


		TEMPERATURE - Product Recipe Extension

			DSTempCtrlRecipe 			: ARRAY [0..iProductRecipeArrayQty] OF DSV3_TempCtrlRecipe;  (* Make it Global so that future can read/write easily*)	

	*)
END_STRUCT
END_TYPE

// ---- DUTs/DS TBD/DS_ArmPnPInOut.TcDUT
TYPE DS_ArmPnPInOut :
STRUCT

	lrHorzLdHookPos : LREAL;
	lrHorzUldHookPos : LREAL;
	ARlrHorzStnHookPos : ARRAY [1..iStnQty] OF LREAL;

	lrHorzLdUnhookPos : LREAL;
	lrHorzUldUnhookPos : LREAL;
	ARlrHorzStnUnhookPos : ARRAY [1..iStnQty] OF LREAL;

	lrVertLdSafeHeightPos : LREAL;
	lrVertUldSafeHeightPos : LREAL;
	ARlrVertStnSafeHeightPos : ARRAY [1..iStnQty] OF LREAL;

	ArlrVertTopPos			: ARRAY [1..iArmQty] OF LREAL;

	lrVertLdDownPos		: LREAL;
	lrVertUldDownPos		: LREAL;
	ARlrVertStnDownPos	: ARRAY [1..iStnQty] OF LREAL;

	ARlrVertStnSlowPullDownPos	: ARRAY [1..iStnQty] OF LREAL;

	lrSlowPullDownPos    : LREAL;
	lrSlowPullUpPos    : LREAL;
	lrSlowPullDownAgitationPos : LREAL;
	lrSlowPullUpAgitationPos : LREAL;

	Fix_VertSpeed	: LREAL;
	Fix_VertAcc		: LREAL;
	Fix_VertDcc		: LREAL;

	Fix_HorzSpeed	: LREAL;
	Fix_HorzAcc		: LREAL;
	Fix_HorzDcc		: LREAL;

	lrSlowPullDownVelo      : LREAL;
	lrSlowPullDownAcc      : LREAL;
	lrSlowPullDownDcc      : LREAL;

	lrSlowPullDown2ndVelo      : LREAL;
	lrSlowPullDown2ndAcc      : LREAL;
	lrSlowPullDown2ndDcc      : LREAL;

	lrSlowPullUpVelo      : LREAL;
	lrSlowPullUpAcc      : LREAL;
	lrSlowPullUpDcc      : LREAL;

	lrSlowPullUp2ndVelo      : LREAL;
	lrSlowPullUp2ndAcc      : LREAL;
	lrSlowPullUp2ndDcc      : LREAL;

END_STRUCT
END_TYPE

// ---- DUTs/DS TBD/DS_BasketInfo.TcDUT
TYPE DS_BasketInfo : (*Full Occupied Byte = 700*)

(*[][][][][][][][][][]----- Basket Information - Attached with Basket -----[][][][][][][][][][]*)

STRUCT
	bAvailibility : BOOL; (* Byte "n" *)
(*	bTimeTrackerEn : BOOL; (* Byte "n+1" *) (***************NEW******************)*)
	sReservedBool : STRING(50); (* Byte "n+2~n+99" *)

	iProductRecipeNo : INT; (* Byte "n+100, n+101" *)
	iProductRecipeStepNo : INT; (* Byte "n+102, n+103" *)
	iStationSeqenceRecipeNo : INT; (* Byte "n+104, n+105" *)
	iPreviousStationNo : INT; (* Byte "n+106, n+107" *)
	iCurrentStationNo : INT; (* Byte "n+108, n+109" *)
(*	iTimeTrackerStepNo : INT; (*Byte "n+110, n+111" *) (***************NEW******************)*)
	sReservedInt : STRING(50); (* Byte "n+112~n+199" *)

	sProgramDescription : STRING(50) ; (* Byte "n+200~n+299" *)
	sProductID : STRING(50); (* Byte "n+300~n+399" *)
	sBarcodeData : STRING(50); (* Byte "n+400~n+499" *)
	sFilePath : STRING(50); (* Byte "n+500~n+599" *)
	sProductQuality : STRING(50); (* Byte "n+600~n+699" *)

END_STRUCT
END_TYPE

// ---- DUTs/DS TBD/DS_BrensonEnclosure.TcDUT
TYPE DS_BrensonEnclosure :
STRUCT
	DSBrensonGenerator : ARRAY [1..iUSGeneratorQty] OF DS_BrensonGenerator;
END_STRUCT
END_TYPE

// ---- DUTs/DS TBD/DS_BrensonGenerator.TcDUT
TYPE DS_BrensonGenerator :
STRUCT
	IN_bUltrasonicStartEn : BOOL;
	IN_bMultiFreqEn :  BOOL;
	IN_iFreqSetPoint :  INT; (* 40/80/120 or 25/50*)
	IN_iTargetPowerPercentSetPoint :  INT; (* 0-100%*)
	IN_lrPowerToAnalogRatio : LREAL; (*Normally for 0-100% is 327.67*)
	IN_lrAnalogInputFineTuneRatio :  LREAL; (*Normally 1, use lower than 1 (example: 0.97) if set to 100% the actual output is greater, use higher than 1 meant the actual output is lesser when you set 100% *)
	IN_lrAnalogOutputFineTuneRatio :  LREAL; (*Normally 1, use lower than 1 (example: 0.97) if set to 100% the actual output is greater, use higher than 1 meant the actual output is lesser when you set 100% *)

	DSBrensonMulFreqSwitching : DS_BrensonMulFreqSwitching;

	OUT_bUltrasonicOnOff :  BOOL;
	OUT_iActualPowerPercentDisplay :  INT; (*Display 0 - 100%*)
	OUT_bFreqSetPointError :  BOOL;

	IN_iPowerAnalogInput  :  INT; (*Link to Terminal*)
	OUT_iPowerAnalogOutput  :  INT; (*Link to Terminal*)

END_STRUCT
END_TYPE

// ---- DUTs/DS TBD/DS_BrensonMulFreqSwitching.TcDUT
TYPE DS_BrensonMulFreqSwitching :
STRUCT
	bFreqSwitchingPB_TS : BOOL;
	bFreqRange4080120En : BOOL;
	bFreqRange2550En : BOOL;
	bDisableMultiFreq80kHz : BOOL;
	iFreqOutput_TS : INT;
END_STRUCT
END_TYPE

// ---- DUTs/DS TBD/DS_ClangsonicGenerator.TcDUT
TYPE DS_ClangsonicGenerator :
STRUCT
	wModbusData : ARRAY [1..iModbusRWQty] OF WORD;
	bModbusWriteEn : ARRAY [1..iModbusRWQty] OF BOOL;

END_STRUCT
END_TYPE

// ---- DUTs/DS TBD/DS_fbGnrProductRecipeMemoryOut.TcDUT
TYPE DS_fbGnrProductRecipeMemoryOut : (*Full Occupied Byte = 1700*)
STRUCT

	bCallCompleted 							: BOOL; (* Byte "n" *)

	bInvalidProductRecipeNoErrHold 		: BOOL; (* Byte "n+1" *)
	bInvalidProductRecipeNoErrPulse		: BOOL; (* Byte "n+2" *)
	bInvalidProductRecipeStepErrHold 		: BOOL; (* Byte "n+3" *)
	bInvalidProductRecipeStepErrPulse		: BOOL; (* Byte "n+4" *)

	bCallUpDownPatternMemoryErr 			: BOOL; (* Byte "n+5" *)
	bCallArmSpeedProfileMemoryErr 		: BOOL; (* Byte "n+6" *)
	bCallPickStationNoErr 					: BOOL; (* Byte "n+7" *)
	bCallTransferStationNoErr 				: BOOL; (* Byte "n+8" *)

	sReservedBool 							: STRING(50); (* Byte "n+9~n+99" *)


	iCalledProductRecipeNo 					: INT; (* Byte "n+100~n+101" *) (*New*)
	iCalledProductRecipeStep				: INT; (* Byte "n+102~n+103" *) (*New*)
	iCallCaseNo 								: INT; (* Byte "n+104~n+105" *)

	sReservedInt 								: STRING(50); (* Byte "n+106~n+199" *)

	sProductRecipeDescription 				: STRING(50);

	DSGnrCalledArmPnpParameter : DSGnr_CalledArmPnpParameter;

END_STRUCT
END_TYPE

// ---- DUTs/DS TBD/DS_fbStationSequenceRecipeCall.TcDUT
TYPE DS_fbStationSequenceRecipeCall : (*Full Occupied Byte = 500*)
STRUCT
	bCallPB: BOOL; (* Byte "n" *)
	bCallCompleted : BOOL; (* Byte "n+1" *)
	bInvalidCallStationSequenceNoHold : BOOL; (* Byte "n+2" *)
	bInvalidCallStationSequenceNoPulse : BOOL; (* Byte "n+3" *)
	sReservedBool : STRING(50); (* Byte "n+4~n+99" *)


	Call_iStationSequenceRecipe : INT; (* Byte "n+100, n+101" *)
	sReservedInt : STRING(50); (* Byte "n+102~n+199" *)


	Call_sSequenceRecipeDescription : STRING(50); (* Byte "n+200~n+299" *)


	Call_DsStationSequenceRecipeMemory : DS_StationSequenceRecipeMemory; (* Byte "n+300 onward" *)





END_STRUCT
END_TYPE

// ---- DUTs/DS TBD/DS_fbStationSequenceRecipeStore.TcDUT
TYPE DS_fbStationSequenceRecipeStore : (*Full Occupied Byte = 500*)
STRUCT

	bCopyPB : BOOL; (* Byte "n" *)
	sReservedBool : STRING(50); (* Byte "n+1~n+99" *)


	iStationSequenceRecipeNo: INT; (* Byte "n+100, n+101" *)	(* 10 sets of Station Sequence Recipe *)
	iCopyToSubRecipeNo : INT; (* Byte "n+102, n+103" *)
	sReservedInt : STRING(50); (* Byte "n+104~n+199" *)


	sStationSequenceRecipeDescription : STRING(50); (* Byte "n+200~n+299" *)  (* Description of Station Sequence Recipe - Naming*)


	DsStationSequenceRecipeMemory : DS_StationSequenceRecipeMemory; (* Byte "n+300 onward" *)






END_STRUCT
END_TYPE

// ---- DUTs/DS TBD/DS_fbStationSubRecipeCall.TcDUT
TYPE DS_fbStationSubRecipeCall : (*Full Occupied Byte = 700*)
STRUCT

	bCallPB: BOOL; (* Byte "n" *)
	bCallCompleted : BOOL; (* Byte "n+1" *)
	bInvalidCallSubRecipeNoHold: BOOL; (* Byte "n+2" *)
	bInvalidCallSubRecipeNoPulse: BOOL; (* Byte "n+3" *)
	sReservedBool : STRING(50); (* Byte "n+4~n+99" *)

	Call_iSubRecipe : INT; (* Byte "n+100, n+101" *)
	sReservedInt : STRING(50); (* Byte "n+102~n+199" *)


	Call_sSubDescription : STRING(50); (* Byte "n+200~n+299" *)


	Call_DsSubRecipeMemory : DS_SubRecipeMemory; (* Byte "n+300 onward" *)






END_STRUCT
END_TYPE

// ---- DUTs/DS TBD/DS_fbStationSubRecipeStore.TcDUT
TYPE DS_fbStationSubRecipeStore : (*Full Occupied Byte = 700*)
STRUCT

	bCopyPB : BOOL; (* Byte "n" *)
	sReservedBool : STRING(50); (* Byte "n+1~n+99" *)


	iSubRecipeNo : INT; (* Byte "n+100, n+101" *) (* 10 sets of Sub Recipe *)
	iCopyToSubRecipeNo : INT; (* Byte "n+102, n+103" *)
	sReservedInt : STRING(50); (* Byte "n+104~n+199" *)


	sSubRecipeDescription : STRING(50); (* Byte "n+200~n+299" *) (* Description of Sub Recipe - Naming*)


	DsSubRecipeMemory : DS_SubRecipeMemory; (* Byte "n+300 onward" *)





END_STRUCT
END_TYPE

// ---- DUTs/DS TBD/DS_fbStnSeqProcessCtrl.TcDUT
TYPE DS_fbStnSeqProcessCtrl : (*Full Occupied Byte = 200*)
STRUCT

	In_bProcessStart 								: BOOL; (* Byte "n" *)
	In_bProcessHalt								: BOOL; (* Byte "n+1" *)
	In_bProcessReset 							: BOOL; (* Byte "n+2" *)

	Out_bProcessCompleted 					: BOOL; (* Byte "n+3" *)
	Out_bProcessInProgressFlag 				: BOOL; (* Byte "n+4" *)
	Out_bProcessHaltFlag 						: BOOL; (* Byte "n+5" *)
	Err_bCallStnSeqRecipeErr 					: BOOL; (* Byte "n+6" *)
	Err_bInvalidProcessStepErr 					: BOOL; (* Byte "n+7" *)

	NIL_sReservedBool 							: STRING(50); (* Byte "n+8~n+99" *)



	Out_iCurrentProcessStep 					: INT; (* Byte "n+100, n+101" *)
	Out_iComConProcessTimeEV 				: INT; (* Byte "n+102, n+103" *)
	Out_iCurrentProcessTime 					: INT; (* Byte "n+104, n+105" *)
	Out_iPreviousProcessTime 					: INT; (* Byte "n+106, n+107" *)
	Out_iStnSeqProcessCaseNo 				: INT; (* Byte "n+108, n+109" *)
	Out_iTotalProcessTimeEV					: INT; (* Byte "n+110, n+111" *)									(* Output - Total Process Elapse Time (DownCounting) (Based Total Time) *)
	Out_ARiCurrentCycle 							: ARRAY [1..iProductRecipeStepArrayQty] OF INT; (* Byte "n+112, n+131" *)
	Out_AR5iCalledTotalProcessTimeSV		: ARRAY [1..5] OF INT;	(* Byte "n+132, n+141" *)					(* Output -  It can accept concurrently 5 different Recipe Total Time based on the Recipe Number defined in AR5iCallTotalTimeRecipeNo*)
	In_AR5iCallTotalTimeRecipeNo				: ARRAY [1..5] OF INT;	(* Byte "n+142, n+151" *)					(* Output -  It can accept concurrently 5 different Recipe Total Time based on the Recipe Number defined in AR5iCallTotalTimeRecipeNo*)

	NIL_sReservedInt 							: STRING(50); (* Byte "n+152~n+199" *)

	Out_DSStnSeqProOutput 					: DS_StnSeqProOutput;
	In_DsStnSeqProInput							: DS_StnSeqProInput;

END_STRUCT
END_TYPE

// ---- DUTs/DS TBD/DS_HMIStationDisplayInfo.TcDUT
TYPE DS_HMIStationDisplayInfo :
STRUCT



	iProductRecipeNo : INT; (*Product Recipe No*)
	iProductRecipeStepNo : INT; (*Product Recipe Step No*)

	iStationSeqenceRecipeNo : INT; (*Station Sequence Recipe No*)
	iStationSequenceRecipeStepNo : INT; (*Current StationSequenceRecipe Step No*)

	iSubRecipeNo : INT; (*Sub Recipe No*)

	iSubRecipeTimeEV : INT; (*Sub recipe Time EV*)
	iTotalProcessTimeEV : INT;(*Process Total Time EV*)


	bStationSequenceProcessStart : BOOL; (*Indicator*)
	bStationSequenceProcessInProgressFlag : BOOL; (*Indicator*)
	bStationSequenceProcessCompleted : BOOL; (*Indicator*)

	bCallStnSeqRecipeErr : BOOL; (*Error Message*)
	bInvalidProcessStepErr : BOOL; (*Error Message*)


	bCallArmSpeedProfileMemoryErr : BOOL; (*Error Message*)

	bCallPickStationNoErr				: BOOL; (*New Error Message*)
	bCallTransferStationNoErr			: BOOL; (*New Error Message*)
	bCallUpDownPatternMemoryErr		: BOOL; (*New Error Message*)
	bInvalidProductRecipeNoErr		: BOOL; (*New Error Message*)
	bInvalidProductRecipeStepErr		: BOOL; (*New Error Message*)

	sErrorMessage : STRING(50);
	sProductRecipeDescription : STRING(50); (*Product Recipe Description*)
	sStationSequenceRecipeDescription : STRING(50); (*StationSequenceRecipeDescription*)
	sStationSubDescription : STRING(50); (*Station Sub Recipe Description*)



END_STRUCT
END_TYPE

// ---- DUTs/DS TBD/DS_HomingSetting.TcDUT
TYPE DS_HomingSetting :
STRUCT

(*Arm Homing*)
(*==================================================*)
	lrArm1HorzHomeVelo 				: LREAL;
	lrArm1HorzHomeAcc 				: LREAL ;
	lrArm1HorzHomeDcc 				: LREAL;
	lrArm1Horz2HomeVelo 			: LREAL;
	lrArm1Horz2HomeAcc 				: LREAL;
	lrArm1Horz2HomeDcc 				: LREAL;

	lrArm1VertHomeVelo 				: LREAL;
	lrArm1VertHomeAcc 				: LREAL;
	lrArm1VertHomeDcc 				: LREAL;
	lrArm1Vert2HomeVelo				: LREAL;
	lrArm1Vert2HomeAcc 				: LREAL;
	lrArm1Vert2HomeDcc 				: LREAL;

	lrArm2HorzHomeVelo 				: LREAL;
	lrArm2HorzHomeAcc 				: LREAL ;
	lrArm2HorzHomeDcc 				: LREAL;
	lrArm2Horz2HomeVelo 			: LREAL;
	lrArm2Horz2HomeAcc 				: LREAL;
	lrArm2Horz2HomeDcc 				: LREAL;

	lrArm2VertHomeVelo 				: LREAL;
	lrArm2VertHomeAcc 				: LREAL;
	lrArm2VertHomeDcc 				: LREAL;
	lrArm2Vert2HomeVelo				: LREAL;
	lrArm2Vert2HomeAcc 				: LREAL;
	lrArm2Vert2HomeDcc 				: LREAL;

	lrArmLifterHomeVelo 				: LREAL;
	lrArmLifterHomeAcc 				: LREAL;
	lrArmLifterHomeDcc 				: LREAL;
	lrArmLifter2HomeVelo				: LREAL;
	lrArmLifter2HomeAcc 				: LREAL;
	lrArmLifter2HomeDcc 				: LREAL;

END_STRUCT
END_TYPE

// ---- DUTs/DS TBD/DS_Inverter.TcDUT
TYPE DS_Inverter :
STRUCT

(*Homing Used*)

	bVertHome_In_HomingSt 								: BOOL;
	bVertHome_In_HomingReset 							: BOOL;
	bVertHome_In_NegativeHomingDirectionEn 				: BOOL;
	bVertHome_In_PositiveHomingDirectionEn 				: BOOL;
	bVertHome_In_HomeSensor 							: BOOL;
	rVertHome_In_HighSpeedHz 							: REAL;
	rVertHome_In_2ndSpeedHz 							: REAL;
	rVertHome_In_DccDelayTimeSec 						: REAL;
	bVertHome_Out_HomeDone 							: BOOL;
	bVertHome_Out_Busy 									: BOOL;
	bVertHome_Out_InvMoveFwd 							: BOOL;
	bVertHome_Out_InvMoveRwd 							: BOOL;
	bVertHome_Out_EncoderValueReset 					: BOOL;
	rVertHome_Out_TargetSpdHz 							: REAL;
	iVertHomeStep										: INT;

	bHorzHome_In_HomingSt 								: BOOL;
	bHorzHome_In_HomingReset 							: BOOL;
	bHorzHome_In_NegativeHomingDirectionEn 				: BOOL;
	bHorzHome_In_PositiveHomingDirectionEn 				: BOOL;
	bHorzHome_In_HomeSensor 							: BOOL;
	rHorzHome_In_HighSpeedHz 							: REAL;
	rHorzHome_In_2ndSpeedHz 							: REAL;
	rHorzHome_In_DccDelayTimeSec 						: REAL;
	bHorzHome_Out_HomeDone 							: BOOL;
	bHorzHome_Out_Busy 								: BOOL;
	bHorzHome_Out_InvMoveFwd 							: BOOL;
	bHorzHome_Out_InvMoveRwd 							: BOOL;
	bHorzHome_Out_EncoderValueReset 					: BOOL;
	rHorzHome_Out_TargetSpdHz 							: REAL;
	iHorzHomeStep										: INT;

(*Jog Used*)

	bJog_InOut_JogEn 									: BOOL;
	bVertJog_In_PositiveJogDirectionSt 						: BOOL;
	bVertJog_In_NegativeJogDirectionSt 					: BOOL;
	rVertJog_In_JogSpeedHz 								: REAL;

	bVertJog_Out_InvMoveFwd 							: BOOL;
	bVertJog_Out_InvMoveRwd 							: BOOL;
	rVertJog_Out_TargetSpdHz 							: REAL;

	bHorzJog_In_PositiveJogDirectionSt 						: BOOL;
	bHorzJog_In_NegativeJogDirectionSt 					: BOOL;
	rHorzJog_In_JogSpeedHz 								: REAL;
	bHorzJog_Out_InvMoveFwd 							: BOOL;
	bHorzJog_Out_InvMoveRwd 							: BOOL;
	rHorzJog_Out_TargetSpdHz 							: REAL;

(* Arm Positioning Signal Control *)

	lrVertFix_PosCfmTolerance								: LREAL;
	lrVertFix_2ndSpdRange								: LREAL;


	lrHorzFix_PosCfmTolerance							: LREAL;
	lrHorzFix_2ndSpdRange								: LREAL;







(* Arm Inv Analog Spd Ctrl*)

	bVert_IASC_Out_JogInProgress 							: BOOL;
	bVert_IASC_Out_HomeInProgress 						: BOOL;
	bVert_IASC_Out_PosInProgress 							: BOOL;
	iVert_Ext_AO_AnalogOutput 							: INT;
	rVert_TS_TargetHzDisplay 								: REAL;


	bHorz_IASC_Out_JogInProgress 						: BOOL;
	bHorz_IASC_Out_HomeInProgress 						: BOOL;
	bHorz_IASC_Out_PosInProgress 						: BOOL;
	iHorz_Ext_AO_AnalogOutput 							: INT;
	rHorz_TS_TargetHzDisplay 							: REAL;


(* General Used*)

	bGen_In_Estop 										: BOOL;
	bGen_In_VertMovementEn								: BOOL;
	bGen_In_HorzMovementEn								: BOOL;


	bVertGen_In_FwdOverTravelSensorNC 					: BOOL;
	bVertGen_In_RwdOverTravelSensorNC 					: BOOL;
	lrVertGen_In_CurrentPos								: LREAL;
	rVertGen_In_HzToRawRatio 							: REAL;
	lrVertGen_InOut_TargetPos								: LREAL;

	bHorzGen_In_FwdOverTravelSensorNC 					: BOOL;
	bHorzGen_In_RwdOverTravelSensorNC 					: BOOL;
	lrHorzGen_In_CurrentPos								: LREAL;
	rHorzGen_In_HzToRawRatio 							: REAL;
	lrHorzGen_InOut_TargetPos							: LREAL;



(* Pos Ctrl Used*)

	bVertPos_In_4StepsEn									: BOOL;
	bVertPos_In_PositioningEn 								: BOOL;
	rVertPos_In_TargetSpdHz								: REAL;
	rVertPos_In_2ndSpdHz									: REAL;
	bVertPos_Out_PositioningDone 							: BOOL;
	bVertPos_Out_PositioningBusy 							: BOOL;
	bVertPos_Out_InvMoveFwd 							: BOOL;
	bVertPos_Out_InvMoveRwd							: BOOL;
	bVertPos_Out_InvMove2ndSpd 							: BOOL;
	rVertPos_Out_TargetSpdHz 							: REAL;


	bHorzPos_In_4StepsEn								: BOOL;
	bHorzPos_In_PositioningEn 							: BOOL;
	rHorzPos_In_TargetSpdHz								: REAL;
	rHorzPos_In_2ndSpdHz								: REAL;
	bHorzPos_Out_PositioningDone 						: BOOL;
	bHorzPos_Out_PositioningBusy 							: BOOL;
	bHorzPos_Out_InvMoveFwd 							: BOOL;
	bHorzPos_Out_InvMoveRwd							: BOOL;
	bHorzPos_Out_InvMove2ndSpd 							: BOOL;
	rHorzPos_Out_TargetSpdHz 							: REAL;


END_STRUCT
END_TYPE

// ---- DUTs/DS TBD/DS_ProminentDosingHMI.TcDUT
TYPE DS_ProminentDosingHMI :
STRUCT
	In_bCalibratePB							: BOOL;
	In_iCalibrateFeed_Pulse					: INT;
	In_iCalibrateTotalVolumeResult_ml			: INT;
	Out_bCalibrateInProgress					: BOOL;
	Out_bCalibrateDone						: BOOL;

	In_rVolumePerPulse_ml 					: REAL; (*Replaced from INT*)
	in_iFirstFillDosing_ml 						: INT;
	In_iVolumePerBasket_ml 					: INT;
	In_iNoOfBasketBetweenAutoDosing 			: INT;
	In_iManualDosingVolume_ml 				: INT;

	In_bResetRemainedDosingVolumePB 		: BOOL;
	Out_bResetRemainedDosingVolumeIndicator 	: BOOL;
	Out_rRemainedDosingVolume_ml 			: REAL; (*Replaced from INT*)

	In_bResetDosingTotalizerPB				: BOOL;
	Out_bResetDosingTotalizerIndicator			: BOOL;
	Out_iDosingTotalizer_Litre 					: INT;
	Out_iDosingTotalizer_ml					: INT;

	Out_iBasketQtyBeforeAutoDosingPV			: INT;

	Out_sStatusMessage						: STRING(50);



END_STRUCT
END_TYPE

// ---- DUTs/DS TBD/DS_SA_Movement.TcDUT
TYPE DS_SA_Movement :
STRUCT

	b_Execute	: BOOL;
	b_Terminate	: BOOL;

	lrZone1StartPos	: LREAL;
	lrZone2StartPos	: LREAL;
	lrZone3StartPos	: LREAL;
	lrZone4StartPos	: LREAL;

	lrZone1EndPos	: LREAL;
	lrZone2EndPos	: LREAL;
	lrZone3EndPos	: LREAL;
	lrZone4EndPos	: LREAL;

	lzZone1EndSpeed	: LREAL;
	lzZone2EndSpeed	: LREAL;
	lzZone3EndSpeed	: LREAL;
	lzZone4EndSpeed	: LREAL;

	lrZone1Speed	: LREAL;
	lrZone1Acc		: LREAL;
	lrZone1Dcc		: LREAL;

	lrZone2Speed	: LREAL;
	lrZone2Acc		: LREAL;
	lrZone2Dcc		: LREAL;

	lrZone3Speed	: LREAL;
	lrZone3Acc		: LREAL;
	lrZone3Dcc		: LREAL;

	lrZone4Speed	: LREAL;
	lrZone4Acc		: LREAL;
	lrZone4Dcc		: LREAL;

	(*Keep this*)
	iLdId			: INT;
	iUldId			: INT;

	Fix_VertSpeed	: LREAL;
	Fix_VertAcc		: LREAL;
	Fix_VertDcc		: LREAL;

	Fix_HorzSpeed	: LREAL;
	Fix_HorzAcc		: LREAL;
	Fix_HorzDcc		: LREAL;

END_STRUCT
END_TYPE

// ---- DUTs/DS TBD/DS_Servo.TcDUT
TYPE DS_Servo :
STRUCT
(*Homing Used*)

	bHome_In_HomingSt 									: BOOL;
	bHome_In_HomingReset 								: BOOL;
	bHome_In_HomeSensor 								: BOOL;
	lrHome_In_HighSpeed	 								: LREAL;
	lrHome_In_HighSpeedAcc	 							: LREAL;
	lrHome_In_HighSpeedDcc	 							: LREAL;
	lrHome_In_2ndSpeed	 								: LREAL;
	lrHome_In_2ndSpeedAcc	 							: LREAL;
	lrHome_In_2ndSpeedDcc	 							: LREAL;
	rHome_In_DccDelayTimeSec 							: REAL;
	bHome_Out_HomeDone 								: BOOL;
	bHome_Out_Busy 									: BOOL;

(*Jog Used*)

	bJog_InOut_JogEn 									: BOOL;
	bJog_In_PositiveJogDirectionSt 							: BOOL;
	bJog_In_NegativeJogDirectionSt 						: BOOL;
	lrJog_In_JogSpeedHz 									: LREAL;
	lrJog_In_JogSpeedAcc 								: LREAL;
	lrJog_In_JogSpeedDcc 								: LREAL;
	bJog_Out_InvMoveFwd 								: BOOL;
	bJog_Out_InvMoveRwd 								: BOOL;

(* Arm Inv Analog Spd Ctrl*)

	bOut_JogInProgress 									: BOOL;
	bOut_HomeInProgress 								: BOOL;
	bOut_PosInProgress 									: BOOL;
	lrOur_RealTimeSpeedDisplay		 					: LREAL;


(* General Used*)

	bGen_In_VertMovementEn								: BOOL;
	bGen_In_HorzMovementEn								: BOOL;
(*	bGen_In_ServoErrorReset								: BOOL;*)

	bGen_In_FwdOverTravelSensorNC 						: BOOL;
	bGen_In_RwdOverTravelSensorNC 						: BOOL;
	lrGen_Out_CurrentPos									: LREAL;

(* Pos Ctrl Used*)

	bPos_In_4StepsEn									: BOOL;
	bPos_In_PositioningEn 								: BOOL;
	bPos_In_Tolerance									: LREAL;
	bPos_Out_PositioningDone 							: BOOL;
	bPos_Out_PositioningBusy 								: BOOL;
	lrPos_In_HighSpeed									: LREAL;
	lrPos_In_Acc											: LREAL;
	lrPos_In_Dcc											: LREAL;

(*	lrPos_In_LowSpeed									: LREAL;*)
(*	Axis_In_Define										: Axis_Ref;*)

(*MC read status *)

	MC_ArmValid											: BOOL;
	MC_ArmBusy											: BOOL;
	MC_ArmError											: BOOL;
	MC_ArmErrorID										: UDINT;
	MC_ArmErrorStop										: BOOL;
	MC_ArmDisable										: BOOL;
	MC_ArmStopping 										: BOOL;
	MC_ArmStandStill										: BOOL;
	MC_ArmDiscreteMotion								: BOOL;
	MC_ArmContinuosMotion								: BOOL;
	MC_ArmSynchronizeMotion								: BOOL;
	MC_ArmHoming										: BOOL;
	MC_ConstantVelocity									: BOOL;
	MC_Acc												: BOOL;
	MC_Dcc												: BOOL;
	MC_Status											: ST_AxisStatus;

END_STRUCT
END_TYPE

// ---- DUTs/DS TBD/DS_StationSequenceRecipeMemory.TcDUT
TYPE DS_StationSequenceRecipeMemory : (*Full Occupied Byte = 200*)
STRUCT

	sReservedBool 				: STRING(50); (* Byte "n+0 ~ n+99" *)

	AR10iStationSubProNo 		: ARRAY [0..iProductRecipeStepArrayQty] OF INT; (* Byte "n100~n+121" *) (* 10 units of SubProcessProgramNo / Steps *)
	AR10iCycle 					: ARRAY [0..iProductRecipeStepArrayQty] OF INT; (* Byte "n+122~n+143" *) (* 10 units of Integer to Store the Cycle needed on the specified Steps. at least "1" *)
	AR10iRepeatFromStepNo 	: ARRAY [0..iProductRecipeStepArrayQty] OF INT; (* Byte "n+144~n+165" *) (* 10 units of Integer to when Cycle repeat, it will repeat from Which Steps  *)
	sReservedInt 					: STRING(50); (* Byte "n+166~n+199" *)




END_STRUCT
END_TYPE

// ---- DUTs/DS TBD/DS_StnSeqProInput.TcDUT
TYPE DS_StnSeqProInput : (*Full Occupied Byte = 200*)

STRUCT
	bProLowLiquidLevel_NC : BOOL; (* Byte "n" *)
	bProRegLiquidLevel_NO : BOOL; (* Byte "n+1" *)
	bProHighLiquidLevel_NO : BOOL; (* Byte "n+1" *)

	bSubLowLiquidLevel_NC : BOOL; (* Byte "n" *)
	bSubRegLiquidLevel_NO : BOOL; (* Byte "n+1" *)
	bSubHighLiquidLevel_NO : BOOL; (* Byte "n+1" *)

	bLowVacuumLevel_NO : BOOL; (* Byte "n+2" *)
	bRegVacuumLevel_NO : BOOL; (* Byte "n+3" *)
	bLowPressureLevel_NO : BOOL; (* Byte "n+4" *)
	bRegPressureLevel_NO : BOOL; (* Byte "n+5" *)
	bExternalActivation_NO : BOOL; (* Byte "n+6" *)
	sReservedBool : STRING(50); (* Byte "n+7~n+99" *)

	iVacuumLevelPV : INT; (* Byte "n+100, n+101" *)
	iPressureLevelPV : INT; (* Byte "n+102, n+103" *)
	iProTankTempLevelPV : INT; (* Byte "n+104, n+105" *)
	iSubTankTempLevelPV : INT; (* Byte "n+106, n+107" *)

	iSlowPullUpPos : INT; (*Used when the station with Slow Pull*)
	iSlowPullDownPos : INT; (*Used when the station with Slow Pull*)

	sReservedInt : STRING(50); (* Byte "n+108~n+199" *)


END_STRUCT
END_TYPE

// ---- DUTs/DS TBD/DS_StnSeqProOutput.TcDUT
TYPE DS_StnSeqProOutput : (*Full Occupied Byte = 200*)
STRUCT
	b1ProTankPump : BOOL; (* Byte "n" *)
	b2ProTankHeater : BOOL; (* Byte "n+1" *)
	b3ProTankBottomUltrasonicA : BOOL; (* Byte "n+2" *)
	b4ProTankBottomUltrasonicB : BOOL; (* Byte "n+3" *)
	b5ProTankBottomUltrasonicC : BOOL; (* Byte "n+4" *)
	b6ProTankSideUltrasonicA : BOOL; (* Byte "n+5" *)
	b7ProTankSideUltrasonicB : BOOL; (* Byte "n+6" *)
	b8SubTankPump : BOOL; (* Byte "n+7" *)
	b9SubTankHeater : BOOL; (* Byte "n+8" *)
	b10Blower : BOOL; (* Byte "n+9" *)
	b11VacuumPump : BOOL; (* Byte "n+10" *)
	b12SlowPull : BOOL; (* Byte "n+11" *)
	b13Instrument2 : BOOL; (* Byte "n+12" *)
	b14Instrument3 : BOOL; (* Byte "n+13" *)
	b15Instrument4 : BOOL; (* Byte "n+14" *)

	b1ActValve1 : BOOL; (* Byte "n+15" *)
	b2ActValve2 : BOOL; (* Byte "n+16" *)
	b3ActValve3 : BOOL; (* Byte "n+17" *)
	b4ActValve4 : BOOL; (* Byte "n+18" *)
	b5ActValve5 : BOOL; (* Byte "n+19" *)
	b6ActValve6 : BOOL; (* Byte "n+20" *)
	b7ActValve7 : BOOL; (* Byte "n+21" *)
	b8ActValve8 : BOOL; (* Byte "n+22" *)
	b9ActValve9 : BOOL; (* Byte "n+23" *)
	b10ActValve10 : BOOL; (* Byte "n+24" *)
	b11ActValve11 : BOOL; (* Byte "n+25" *)
	b12ActValve12 : BOOL; (* Byte "n+26" *)
	b13ActValve13 : BOOL; (* Byte "n+27" *)
	b14ActValve14 : BOOL; (* Byte "n+28" *)
	b15ActValve15 : BOOL; (* Byte "n+29" *)
	b16ActValve16 : BOOL; (* Byte "n+30" *)
	b17ActValve17 : BOOL; (* Byte "n+31" *)
	b18ActValve18 : BOOL; (* Byte "n+32" *)
	b19ActValve19 : BOOL; (* Byte "n+33" *)
	b20ActValve20 : BOOL; (* Byte "n+34" *)

	b16EnProTankChangeTemp : BOOL; (* Byte "n+35" *) (*New*)
	b17EnSubTankChangeTemp : BOOL; (* Byte "n+36" *) (*New*)

	sReservedBool : STRING(50); (* Byte "n+37~n+99" *)

